METHOD FB_init : BOOL
VAR_INPUT
	bInitRetains : BOOL; // if TRUE, the retain variables are initialized (warm start / cold start)
	bInCopyCode : BOOL;  // if TRUE, the instance afterwards gets moved into the copy code (online change)
	stPTOStepperRef : POINTER TO ST_PTOStepperRef;
END_VAR
THIS^.pPTOStepperRef := stPTOStepperRef;
END_METHOD

PROPERTY P_bError : BOOL
GET
END_GET
END_PROPERTY

PROPERTY P_bIsActive : BOOL
GET
END_GET
END_PROPERTY

PROPERTY P_bIsLocked : BOOL
GET
P_bIsLocked := TRUE;
END_GET
END_PROPERTY

PROPERTY P_pPTOStepperRef : POINTER TO ST_PTOStepperRef
GET
P_pPTOStepperRef := pPTOStepperRef;
END_GET
END_PROPERTY

END_FUNCTION_BLOCK

// ---- Hardware/PTOStepper/FB_PTOStepperRotate.TcPOU
FUNCTION_BLOCK FB_PTOStepperRotate
VAR_INPUT
	bExecute	: BOOL;
	bStop		: BOOL;
	bCCW		: BOOL;	//Gegen Uhrzeiger
	nSpeed		: UINT;	//Steps/sec
END_VAR
VAR_OUTPUT
	bBusy		: BOOL;
END_VAR
VAR_IN_OUT
	pPTOStepperRef : POINTER TO ST_PTOStepperRef;
END_VAR
VAR
	nSpeedIntern : INT;
	nState : USINT;
END_VAR

IF bExecute THEN
	CASE nState OF
		0:	//Prepare
			IF bStop THEN
				RETURN;
			END_IF
			bBusy := TRUE;
			IF bCCW THEN
				nSpeedIntern := UINT_TO_INT(nSpeed);
			ELSE
				nSpeedIntern := -UINT_TO_INT(nSpeed);
			END_IF
			MEMCPY(ADR(pPTOStepperRef^.nFrequencyValue),ADR(nSpeedIntern),2);
			nState := 1;
			
		1:	//Waiting for stop
			IF bStop THEN
				pPTOStepperRef^.nFrequencyValue := 0;
				nState := 80;
				bBusy := FALSE;
			END_IF
	END_CASE
ELSE
	nState := 0;
	bBusy := FALSE;	
END_IF

END_FUNCTION_BLOCK

// ---- Hardware/PTOStepper/FB_PTOStepperMoveRel.TcPOU
FUNCTION_BLOCK FB_PTOStepperMoveRel
VAR_INPUT
	bExecute	: BOOL;
	bStop		: BOOL;
	nSteps		: INT;
	nSpeed		: UINT;	//Steps/sec	
END_VAR
VAR_OUTPUT
	bBusy		: BOOL;
END_VAR
VAR_IN_OUT
	pPTOStepperRef : POINTER TO ST_PTOStepperRef;	
END_VAR
VAR
	nState : USINT;
	nSpeedIntern: INT;
END_VAR

IF bExecute THEN
	CASE nState OF
		0:	//Prepare
			IF bStop THEN
				RETURN;
			END_IF
			
			bBusy := TRUE;
			IF nSteps < 0 THEN
				//CCW Drehung -> muss Richtung "0" drehen -> auf Counter "0" oder Counter underflow abfragen
				pPTOStepperRef^.nSetCounterValue := INT_TO_UINT(ABS(nSteps));
				nSpeedIntern := -UINT_TO_INT(nSpeed);
			ELSIF nSteps > 0 THEN
				//CW Drehung -> muss Richtung "0" drehen -> auf Counter >= SetCounter oder Counter overflow abfragen
				pPTOStepperRef^.nSetCounterValue := 0;
				nSpeedIntern := UINT_TO_INT(nSpeed);
			ELSE
				bBusy := FALSE;
				nState := 80;
				RETURN;
			END_IF
			pPTOStepperRef^.bSetCounter := TRUE;
			nState := 1;
			
		1:	//Start
			IF bStop THEN
				bBusy := FALSE;
				nState := 80;
				RETURN;
			END_IF
			IF pPTOStepperRef^.nSetCounterValue = pPTOStepperRef^.nCountervalue THEN
				pPTOStepperRef^.bSetCounter := FALSE;
				MEMCPY(ADR(pPTOStepperRef^.nFrequencyValue),ADR(nSpeedIntern),2);
				nState := 2;
			END_IF
			
		2:	//Waiting for target reached
			IF bStop OR
					 	//CCW Drehung -> abwärts zählen -> auf Counter "0" oder Counter underflow abfragen
						((nSteps < 0) AND ((pPTOStepperRef^.nCountervalue = 0) OR pPTOStepperRef^.bCounterUnderflow))
					 OR
					 	//CW Drehung -> aufwärts zählen -> auf Counter >= SetCounter oder Counter overflow abfragen
						((nSteps > 0) AND ((pPTOStepperRef^.nCountervalue >= INT_TO_UINT(ABS(nSteps))) OR pPTOStepperRef^.bCounterUnderflow))THEN
						
				pPTOStepperRef^.nFrequencyValue := 0;
				nState := 3;
			END_IF
			
		3:	//Wartezyklus
			bBusy := FALSE;
	END_CASE
ELSE
	nState := 0;
	bBusy := FALSE;
END_IF

END_FUNCTION_BLOCK

// ---- Hardware/MultiZ/Heater/FB_MzHeaterControl.TcPOU
FUNCTION_BLOCK FB_MzHeaterControl
VAR_INPUT
	bExecute 		: BOOL;
	nTempZone1		: UINT;		//Solltemperatur Heizzone 1
	nTempZone2		: UINT;		//Solltemperatur Heizzone 2
	nTempZone3		: UINT;		//Solltemperatur Heizzone 3
	bHeatingOn		: BOOL;		//Ein/Aus
END_VAR
VAR_OUTPUT
	bBusy : BOOL;
	bError : BOOL;
	nErrorId : ERRORID;	
END_VAR
VAR_IN_OUT
	pFbHeaterRef : POINTER TO FB_MZHeaterRef;
END_VAR
VAR
	fbSdoWrite		: FB_SDO_WRITE;
	fbSdoRead		: FB_SDO_Read;
	nState 			: USINT;
	nStateNext		: USINT;
END_VAR

IF pFbHeaterRef = 0 THEN
	RETURN;
END_IF

IF bExecute THEN
	IF nState = 0 THEN //Solltemperatur Zone 1 senden
		bBusy := TRUE;
		IF NOT bHeatingOn THEN	//keine Temperaturen senden
			nState := 3;
		ELSE
			pFbHeaterRef^.P_nTemp1Setpoint := nTempZone1;
			fbSdoWrite.nIndex := cTempSetPoint.nIndex;
			fbSdoWrite.nSubIndex := pFbHeaterRef^.nChannel;
			fbSdoWrite.nDataLength := cTempSetPoint.nLength;
			fbSdoWrite.nData := UINT_TO_DINT(nTempZone1);
			nState := 10;
			IF pFbHeaterRef^.pMultiZRef^.P_bLegacy THEN	//Heizzone2 und 3 nur bei Firmware ab V1.10.xx
				nStateNext := 3;
			ELSE
				nStateNext := 1;
			END_IF
		END_IF
	END_IF
	
	IF nState = 1 THEN //Solltemperatur Zone 2 senden
		fbSdoWrite.nIndex := cTempSetPoint2.nIndex;
		fbSdoWrite.nSubIndex := pFbHeaterRef^.nChannel;
		fbSdoWrite.nDataLength := cTempSetPoint2.nLength;
		fbSdoWrite.nData := UINT_TO_DINT(nTempZone2);
		nState := 10;
		nStateNext := 2;
	END_IF

	IF nState = 2 THEN //Solltemperatur Zone 3 senden
		fbSdoWrite.nIndex := cTempSetPoint3.nIndex;
		fbSdoWrite.nSubIndex := pFbHeaterRef^.nChannel;
		fbSdoWrite.nDataLength := cTempSetPoint3.nLength;
		fbSdoWrite.nData := UINT_TO_DINT(nTempZone3);
		nState := 10;
		nStateNext := 3;
	END_IF
	
	IF nState = 3 THEN //On/Off senden
		fbSdoWrite.nIndex := cHeatingOn.nIndex;
		fbSdoWrite.nSubIndex := pFbHeaterRef^.nChannel;
		fbSdoWrite.nDataLength := cHeatingOn.nLength;
		fbSdoWrite.nData := BOOL_TO_DINT(bHeatingOn);
		nState := 10;
		IF pFbHeaterRef^.P_bHeaterDetected THEN
			nStateNext := 80;
		ELSE
			nStateNext := 20;
		END_IF
		
	END_IF
	
	IF nState = 10 THEN
		fbSdoWrite(sADSNetID:= pFbHeaterRef^.pMultiZRef^.P_sAdsNetId, nPortNr:= pFbHeaterRef^.pMultiZRef^.P_nAdsPort, bExecute:= TRUE);		
		IF NOT fbSdoWrite.bBusy THEN
			IF fbSdoWrite.bError THEN
				bError := TRUE;
				bBusy := FALSE;
				nErrorId := fbSdoWrite.nAdsErrorId;
				nState := 99;
			ELSE
				nState := nStateNext;
				IF nState = 80 THEN
					bBusy := FALSE;
				END_IF
			END_IF
			fbSdoWrite(bExecute:= FALSE);
		END_IF
	ELSIF nState = 20 THEN //Das HeaterExist wird nur ausgelesen, wenn es nicht vorher schon in A_PrepareAxis im FB_MultiZRef erfolgt ist.
		//Dieser Fall tritt ein, wenn der Heizer später erst angesteckt wurde (Kartuschen-Halter und Piezo-Pipetten)
		fbSdoRead(sADSNetID:= pFbHeaterRef^.pMultiZRef^.P_sAdsNetId, nPortNr:= pFbHeaterRef^.pMultiZRef^.P_nAdsPort, nIndex:= cHeaterExist.nIndex, 
					nSubIndex:= pFbHeaterRef^.nChannel,	nDataLength:= cHeaterExist.nLength, bExecute:= TRUE);
		IF NOT fbSdoRead.bBusy THEN
			IF fbSdoRead.bError THEN
				bError := TRUE;
				bBusy := FALSE;
				nErrorId := fbSdoRead.nAdsErrorId;
				nState := 99;
			ELSE
				pFbHeaterRef^.P_bHeaterDetected := DINT_TO_BOOL(fbSdoRead.nData);
				nState := 80;
				bBusy := FALSE;
			END_IF
			fbSdoRead(bExecute:= FALSE);
		END_IF
	END_IF
ELSE
	nState := 0;
	bError := FALSE;
	nErrorId := 0;
END_IF

END_FUNCTION_BLOCK

// ---- Objects/Tools/FB_PassivPip.TcPOU
FUNCTION_BLOCK FB_PassivPip EXTENDS FB_GCodeTool IMPLEMENTS I_UsingDryPad, I_Dispenser
VAR_INPUT
END_VAR
VAR_OUTPUT
END_VAR
VAR
	//SpecProperties
	nDiluterObjId		: UINT;
	pDiluter			: POINTER TO FB_Diluter;
	pDiluter3Inputs		: POINTER TO FB_Diluter3Inputs;
	nDrypadArea			: USINT;
	tDryTime			: TIME;
	nDispFlowFix		: DINT;	//wird für das Dispensen benutzt, wenn Tool am HybridDispenser oder M127 (UniDispense)

	//****************************************Aktionvariablen****************************************************
	stActionDataSpec	: ST_ActionData;
	
	//Action: "Aspirate"
	bAspirate			: BOOL;
	nStateA_Aspirate	: USINT;
	nQuantity			: DINT;
	nFlow				: DINT;
	
	//Action: "Dispense"
	bDispense			: BOOL;
	nStateA_Dispense	: USINT;
	nDilInput			: USINT;
	bEndless			: BOOL;
	
	//Action: "DilMovePlunger"
	bDilMovePlunger		: BOOL;
	nStateA_DilMovePlunger	: USINT;
	nDilMovePlungerPos	: DINT;
	nDilMovePlungerSpeed: DINT;
	nDilMovePlungerValve: DINT;
	
	
	//Action: "Mix"
	bMix				: BOOL;
	nStateA_Mix			: USINT;
	nFlowAsp			: DINT;
	nFlowDisp			: DINT;
	nMixRepeats			: UINT;
	nCurrMixRepeats		: UINT;
	tMixDelay1			: TIME; //Delay zwischen Asp und Disp
	tMixDelay2			: TIME; //Delay nach jedem Zyklus
	timerMix			: TON;
	
	//Action: "Eject"
	bEject				: BOOL;
	nStateA_Eject		: USINT;
	fbMultiZTipEjector	: FB_MultiZTipEjector;
	
END_VAR

IF eCurrentState = E_MachineState.MACHINESTATE_Active THEN
	
	IF bAspirate THEN
		A_Aspirate();
		IF nStateA_Aspirate >= 80 THEN
			IF nStateA_Aspirate >= 99 THEN
				fbErrorList.M_Add(stError);
				bError := TRUE;	
			END_IF
			bAspirate := FALSE;
			nStateA_Aspirate := 0;
			M_RemoveListEntry(nSearchValue:= E_Action.ACTION_Aspirate);
		END_IF
	END_IF

	IF bDispense THEN
		A_Dispense();
		IF nStateA_Dispense >= 80 THEN
			IF nStateA_Dispense >= 99 THEN
				stError.Cmd := E_Action.ACTION_Dispense;
				fbErrorList.M_Add(stError);
				bError := TRUE;	
			END_IF
			bDispense := FALSE;
			nStateA_Dispense := 0;
			M_RemoveListEntry(nSearchValue:= E_Action.ACTION_Dispense);
		END_IF
	END_IF
	
	IF bMix THEN
		A_Mix();
		IF nStateA_Mix >= 80 THEN
			IF nStateA_Mix >= 99 THEN
				stError.Cmd := E_Action.ACTION_Mix;
				fbErrorList.M_Add(stError);
				bError := TRUE;	
			END_IF
			bMix := FALSE;
			nStateA_Mix := 0;
			M_RemoveListEntry(nSearchValue:= E_Action.ACTION_Mix);
		END_IF
	END_IF
	
	IF bEject THEN
		A_Eject();
		IF nStateA_Eject >= 80 THEN
			IF nStateA_Eject >= 99 THEN
				stError.Cmd := E_Action.ACTION_Eject;
				fbErrorList.M_Add(stError);
				bError := TRUE;	
			END_IF
			bEject := FALSE;
			nStateA_Eject := 0;
			M_RemoveListEntry(nSearchValue:= E_Action.ACTION_Eject);
		END_IF
	END_IF
	
	IF bDilMovePlunger THEN
		A_DilMovePlunger();
		IF nStateA_DilMovePlunger >= 80 THEN
			IF nStateA_DilMovePlunger >= 99 THEN
				stError.Cmd := E_Action.ACTION_DilMovePlunger;
				fbErrorList.M_Add(stError);
				bError := TRUE;	
			END_IF
			bDilMovePlunger := FALSE;
			nStateA_DilMovePlunger := 0;
			M_RemoveListEntry(nSearchValue:= E_Action.ACTION_DilMovePlunger);
		END_IF
	END_IF

END_IF

SUPER^();	//FB_MzTool aufrufen

aObjProcData[nNotifyId] := stProcessData;
stProcessData.n32Data[7] := BOOL_TO_DINT(bAspirate OR bDispense);

ACTION A_Aspirate:
IF pDiluter^.P_bError THEN
	stError.ErrorId := pDiluter^.P_nErrorId;
	stError.POUState := nStateA_Aspirate;
	nStateA_Aspirate := 99;
END_IF

CASE nStateA_Aspirate OF
	0:	MEMSET(ADR(stActionDataSpec),0,SIZEOF(stActionDataSpec));
		stActionDataSpec.eAction := E_Action.ACTION_DilPump;
		stActionDataSpec.aParams[1] := E_DilPumpMode.MODE_Suck;
		stActionDataSpec.aParams[2] := nQuantity; 
		stActionDataSpec.aParams[3] := nFlow;
		//stActionDataSpec.aParams[4]  //ReloadSpeed wird von DilConfig übernommen
		(*Beim normalen Diluter wird ValvePosReload aus der DilConfig übernommen, beim Diluter3Inputs wird
		die ValvePos über die InputNr ermittelt.*)
		IF pDiluter3Inputs > 0 THEN
			stActionDataSpec.aParams[6] := pDiluter3Inputs^.M_GetValvePosInput(nDilInput);
		END_IF
		
		stError.ErrorId := pDiluter^.M_ExeAction(stActionDataSpec);
		IF stError.ErrorId > 0 THEN
			stError.POUState := nStateA_Aspirate;
			nStateA_Aspirate := 99;
		ELSE
			nStateA_Aspirate := 1;	
		END_IF
		
	1:	//Warten bis Aspiration fertig
		IF NOT pDiluter^.M_GetActionBusy(E_Action.ACTION_DilPump) THEN
			nStateA_Aspirate := 80;
		END_IF
		
	70:	//Abbrechen
		MEMSET(ADR(stActionDataSpec),0,SIZEOF(stActionDataSpec));
		stActionDataSpec.eAction := E_Action.ACTION_Stop;
		
		pDiluter^.M_ExeAction(stActionDataSpec);
		nStateA_Aspirate := 71;
		
	71:	
		IF NOT pDiluter^.P_bBusy THEN
			nStateA_Aspirate := 80;
		END_IF
END_CASE

//Errorhandling
IF nStateA_Aspirate = 99 THEN
	stError.Cmd := E_Action.ACTION_Aspirate;
	stError.POU := E_POU.POU_FB_PassivPip;
	stError.POUAction := E_POUACT.POUACT_A_Aspirate;
	fbErrorList.M_Add(stError);
END_IF
END_ACTION

ACTION A_DilMovePlunger:
IF pDiluter^.P_bError THEN
	stError.ErrorId := pDiluter^.P_nErrorId;
	stError.POUState := nStateA_DilMovePlunger;
	nStateA_DilMovePlunger := 99;
END_IF

CASE nStateA_DilMovePlunger OF
	0:	MEMSET(ADR(stActionDataSpec),0,SIZEOF(stActionDataSpec));
		stActionDataSpec.eAction := E_Action.ACTION_DilMovePlunger;
		stActionDataSpec.aParams[1] := nDilMovePlungerPos;
		stActionDataSpec.aParams[2] := nDilMovePlungerSpeed;
		stActionDataSpec.aParams[3] := nDilMovePlungerValve;
		stError.ErrorId := pDiluter^.M_ExeAction(stActionDataSpec);
		IF stError.ErrorId > 0 THEN
			nStateA_DilMovePlunger := 99;
		ELSE
			nStateA_DilMovePlunger := 1;	
		END_IF
	
	1:	IF NOT pDiluter^.M_GetActionBusy(E_Action.ACTION_DilMovePlunger) THEN
			nStateA_DilMovePlunger := 80;
		END_IF
 		
	70: //Abrechen
		MEMSET(ADR(stActionDataSpec),0,SIZEOF(stActionDataSpec));
		stActionDataSpec.eAction := E_Action.ACTION_Stop;
		
		pDiluter^.M_ExeAction(stActionDataSpec);
		nStateA_DilMovePlunger := 71;
		
	71:	IF NOT pDiluter^.P_bBusy THEN
			nStateA_DilMovePlunger := 80;
		END_IF	
END_CASE

//Errorhandling
IF nStateA_DilMovePlunger = 99 THEN
	stError.Cmd := E_Action.ACTION_DilMovePlunger;
	stError.POU := E_POU.POU_FB_PassivPip;
	stError.POUAction := E_POUACT.POUACT_A_MovePlunger;
	fbErrorList.M_Add(stError);
END_IF
END_ACTION

ACTION A_Dispense:
IF pDiluter^.P_bError THEN
	stError.ErrorId := pDiluter^.P_nErrorId;
	stError.POUState := nStateA_Dispense;
	nStateA_Dispense := 99;
END_IF

CASE nStateA_Dispense OF
	0:	MEMSET(ADR(stActionDataSpec),0,SIZEOF(stActionDataSpec));
		stActionDataSpec.eAction := E_Action.ACTION_DilPump;
		stActionDataSpec.aParams[1] := E_DilPumpMode.MODE_Press;
		stActionDataSpec.aParams[2] := nQuantity; 
		stActionDataSpec.aParams[3] := nFlow;
		//stActionDataSpec.aParams[4]  //ReloadSpeed wird von DilConfig übernommen
		(*Beim normalen Diluter wird ValvePosReload aus der DilConfig übernommen, beim Diluter3Inputs wird
		die ValvePos über die InputNr ermittelt.*)
		IF pDiluter3Inputs > 0 THEN
			stActionDataSpec.aParams[6] := pDiluter3Inputs^.M_GetValvePosInput(nDilInput);
		END_IF
		stActionDataSpec.aParams[7] := BOOL_TO_DINT(bEndless);
		bEndless := FALSE;
		
		stError.ErrorId := pDiluter^.M_ExeAction(stActionDataSpec);
		IF stError.ErrorId > 0 THEN
			stError.POUState := nStateA_Dispense;
			nStateA_Dispense := 99;
		ELSE
			nStateA_Dispense := 1;	
		END_IF
		
	1:	//Warten bis Dispensen fertig
		IF NOT pDiluter^.M_GetActionBusy(E_Action.ACTION_DilPump) THEN
			nStateA_Dispense := 80;
		END_IF
		
	70:	//Abbrechen
		MEMSET(ADR(stActionDataSpec),0,SIZEOF(stActionDataSpec));
		stActionDataSpec.eAction := E_Action.ACTION_Stop;
		
		pDiluter^.M_ExeAction(stActionDataSpec);
		nStateA_Dispense := 71;
		
	71:	
		IF NOT pDiluter^.P_bBusy THEN
			nStateA_Dispense := 80;
		END_IF
END_CASE

//Errorhandling
IF nStateA_Dispense = 99 THEN
	stError.Cmd := E_Action.ACTION_Dispense;
	stError.POU := E_POU.POU_FB_PassivPip;
	stError.POUAction := E_POUACT.POUACT_A_Dispense;
	fbErrorList.M_Add(stError);
END_IF
END_ACTION

ACTION A_Eject:
fbMultiZTipEjector(pfbZAxisRef:= pZAxisRef, bExecute:= TRUE);

IF NOT fbMultiZTipEjector.bBusy THEN
	IF fbMultiZTipEjector.bError THEN
		stError.Cmd := E_Action.ACTION_Eject;
		stError.ErrorId := fbMultiZTipEjector.nErrorId;
		stError.POUState := nStateA_Eject;
		stError.POU := E_POU.POU_FB_PassivPip;
		stError.POUAction := E_POUACT.POUACT_A_Eject;
		fbErrorList.M_Add(stError);
		nStateA_Eject := 99;
	ELSE
		nStateA_Eject := 80;
	END_IF
	fbMultiZTipEjector(bExecute:= FALSE);
END_IF
END_ACTION

ACTION A_Mix:
IF pDiluter^.P_bError THEN
	stError.ErrorId := pDiluter^.P_nErrorId;
	stError.POUState := nStateA_Mix;
	nStateA_Mix := 99;
END_IF

CASE nStateA_Mix OF
	0:	//Aspirieren
		MEMSET(ADR(stActionDataSpec),0,SIZEOF(stActionDataSpec));
		stActionDataSpec.eAction := E_Action.ACTION_DilPump;
		stActionDataSpec.aParams[1] := E_DilPumpMode.MODE_Suck;
		stActionDataSpec.aParams[2] := nQuantity; 
		stActionDataSpec.aParams[3] := nFlowAsp;
		//stActionDataSpec.aParams[4]  //ReloadSpeed wird von DilConfig übernommen
		(*Beim normalen Diluter wird ValvePosReload aus der DilConfig übernommen, beim Diluter3Inputs wird
		die ValvePos über die InputNr ermittelt.*)
		IF pDiluter3Inputs > 0 THEN
			stActionDataSpec.aParams[6] := pDiluter3Inputs^.M_GetValvePosInput(nDilInput);
		END_IF
		
		stError.ErrorId := pDiluter^.M_ExeAction(stActionDataSpec);
		IF stError.ErrorId > 0 THEN
			stError.POUState := nStateA_Mix;
			nStateA_Mix := 99;
		ELSE
			nStateA_Mix := 1;	
		END_IF
		
	1:	//Aspirieren fertig?
		IF NOT pDiluter^.M_GetActionBusy(E_Action.ACTION_DilPump) THEN
			timerMix(IN:= TRUE, PT:= tMixDelay1);
			nStateA_Mix := 2;
		END_IF
		
	2:	//Timer?
		timerMix();
		IF timerMix.Q THEN
			timerMix(IN:= FALSE);
			nStateA_Mix := 3;
		END_IF
		
	3:	//Dispensen
		MEMSET(ADR(stActionDataSpec),0,SIZEOF(stActionDataSpec));
		stActionDataSpec.eAction := E_Action.ACTION_DilPump;
		stActionDataSpec.aParams[1] := E_DilPumpMode.MODE_Press;
		stActionDataSpec.aParams[2] := nQuantity; 
		stActionDataSpec.aParams[3] := nFlowDisp;
		//stActionDataSpec.aParams[4]  //ReloadSpeed wird von DilConfig übernommen
		(*Beim normalen Diluter wird ValvePosReload aus der DilConfig übernommen, beim Diluter3Inputs wird
		die ValvePos über die InputNr ermittelt.*)
		IF pDiluter3Inputs > 0 THEN
			stActionDataSpec.aParams[6] := pDiluter3Inputs^.M_GetValvePosInput(nDilInput);
		END_IF
		
		
		stError.ErrorId := pDiluter^.M_ExeAction(stActionDataSpec);
		IF stError.ErrorId > 0 THEN
			stError.POUState := nStateA_Mix;
			nStateA_Mix := 99;
		ELSE
			nStateA_Mix := 4;
		END_IF
		
	4:	//Dispensen fertig?
		IF NOT pDiluter^.M_GetActionBusy(E_Action.ACTION_DilPump) THEN
			nCurrMixRepeats := nCurrMixRepeats + 1;
			IF nCurrMixRepeats = nMixRepeats THEN
				nStateA_Mix := 80;
			ELSE
				timerMix(IN:= TRUE, PT:= tMixDelay2);
				nStateA_Mix := 5;
			END_IF
		END_IF
		
	5:	//Timer?
		timerMix();
		IF timerMix.Q THEN
			timerMix(IN:= FALSE);
			nStateA_Mix := 0;
		END_IF

	70:	//Abbrechen
		timerMix(IN:= FALSE);
		MEMSET(ADR(stActionDataSpec),0,SIZEOF(stActionDataSpec));
		stActionDataSpec.eAction := E_Action.ACTION_Stop;
		pDiluter^.M_ExeAction(stActionDataSpec);
		nStateA_Mix := 71;
		
	71:	IF NOT pDiluter^.P_bBusy THEN
			nStateA_Mix := 80;
		END_IF		
END_CASE

//Errorhandling
IF nStateA_Mix = 99 THEN
	stError.Cmd := E_Action.ACTION_Mix;
	stError.POU := E_POU.POU_FB_PassivPip;
	stError.POUAction := E_POUACT.POUACT_A_Mix;
	fbErrorList.M_Add(stError);
END_IF
END_ACTION

ACTION A_Reset:
//Ist noch eine Aktion aktiv?
IF nStateA_ResetSpec = 0 THEN 
	IF bAspirate THEN
		bAspirate := FALSE;
		nStateA_Aspirate := 0;
	END_IF

	IF bDispense THEN
		bDispense := FALSE;
		nStateA_Dispense := 0;
	END_IF
	
	IF bEject THEN
		bEject := FALSE;
		nStateA_Eject := 0;
	END_IF
	
	nStateA_ResetSpec := 80;
END_IF

SUPER^.A_Reset();
END_ACTION

ACTION A_Stop:
IF nStateA_Stop = 0 THEN
	
	IF bAspirate AND nStateA_Aspirate < 70 THEN
		nStateA_Aspirate := 70;
	END_IF
	
	IF bDispense AND nStateA_Dispense < 70 THEN
		nStateA_Dispense := 70;
	END_IF
	
	IF bMix AND nStateA_Mix < 70 THEN
		nStateA_Mix := 70;
	END_IF
	
	nStateA_Stop := 1;
END_IF

SUPER^.A_Stop();
END_ACTION

METHOD FB_init : BOOL
VAR_INPUT
	bInitRetains : BOOL; // if TRUE, the retain variables are initialized (warm start / cold start)
	bInCopyCode : BOOL;  // if TRUE, the instance afterwards gets moved into the copy code (online change)
END_VAR
eObjectType := E_ObjectType.OBJECTTYPE_PassivPip;
eObjectGroup := E_ObjectGroup.OBJECTGROUP_MzTool OR E_ObjectGroup.OBJECTGROUP_Device;
END_METHOD

METHOD M_AddChild : ERRORID
VAR_INPUT
	pObject : POINTER TO FB_Object;
	nSlotNr	: UINT;
	nIndex 	: INT;
END_VAR
//PassivePip kann folgende Objekt-Typen aufnehmen
//Needle, Tip, Nozzle
IF pObject > 0 THEN
	IF pObject^.P_eObjectType = E_ObjectType.OBJECTTYPE_Needle OR
		pObject^.P_eObjectType = E_ObjectType.OBJECTTYPE_Nozzle OR
		pObject^.P_eObjectType = E_ObjectType.OBJECTTYPE_Tip THEN
		M_AddChild := SUPER^.M_AddChild(pObject,nSlotNr,nIndex);
	ELSE
		M_AddChild := E_ErrorIdObjMgmt.ERRORID_InvalidParentObject;
	END_IF
ELSE
	M_AddChild := E_ErrorIdObjMgmt.ERRORID_InvalidParentObject;
END_IF
END_METHOD

METHOD M_CancelAction
VAR_INPUT
	eAction : E_Action;
END_VAR
CASE eAction OF
	E_Action.ACTION_Aspirate:
		IF bAspirate AND nStateA_Aspirate < 70 THEN
			nStateA_Aspirate := 70;
		END_IF
	E_Action.ACTION_Dispense:
		IF bDispense AND nStateA_Dispense < 70 THEN
			nStateA_Dispense := 70;
		END_IF
	E_Action.ACTION_Mix:
		IF bMix AND nStateA_Mix < 70 THEN
			nStateA_Mix := 70;
		END_IF	
ELSE
	SUPER^.M_CancelAction(eAction);
END_CASE
END_METHOD

METHOD M_CheckAction : ERRORID
VAR_INPUT
	refActionData 	: REFERENCE TO ST_ActionData;
	pCorrelObject	: POINTER TO FB_Object;
END_VAR

VAR
	pTarget : POINTER TO FB_TargetBase;
	pRack	: POINTER TO FB_Rack;
	pSlot	: POINTER TO FB_PieceSlot;	
END_VAR
CASE refActionData.eAction OF
	E_Action.ACTION_GetPipSample,
	E_Action.ACTION_MeasureTool,
	E_Action.ACTION_Dispense, //BasicAction für ActionOnArray
	E_Action.ACTION_Aspirate, //BasicAction für ActionOnArray
	E_Action.ACTION_Mix, //BasicAction für ActionOnArray
	E_Action.ACTION_TeachTarget:
		RETURN;
	E_Action.ACTION_WashTool:
		//Washmode checken
		IF refActionData.aParams[2] = E_WashMode.MODE_WashInside THEN
			M_CheckAction := M_CheckBottles();
		ELSIF refActionData.aParams[2] = E_WashMode.MODE_WashOutside THEN
			;
		ELSIF refActionData.aParams[2] = E_WashMode.MODE_WashInOutside THEN
			M_CheckAction := M_CheckBottles();
		ELSIF refActionData.aParams[2] = E_WashMode.MODE_DryOutside THEN
			;
		ELSE
			M_CheckAction := E_ErrorIdCmd.ERRORID_InvalidWashMode;	
		END_IF
	E_Action.ACTION_InsertTool:
		//PassivPip darf nur in offene Vials eintauchen
		//-> Target muss also ein VialRack sein (Reaktor nicht möglich, da Pip nicht von der Tiefe hinein passt)
		pTarget := pCorrelObject;
		IF pTarget > 0 THEN
			IF (pTarget^.P_eObjectGroup AND E_ObjectGroup.OBJECTGROUP_Rack) = E_ObjectGroup.OBJECTGROUP_Rack THEN
				pRack := pTarget;
				pSlot := pRack^.M_GetSlot(DINT_TO_UINT(refActionData.aParams[2]));
				IF pSlot > 0 THEN
					IF pSlot^.P_pPiece = 0 THEN
						M_CheckAction := E_ErrorIdCmd.ERRORID_NoPieceInSlot;
						RETURN;
					ELSIF NOT (pSlot^.P_pPiece^.P_eObjectType = E_ObjectType.OBJECTTYPE_Vial OR pSlot^.P_pPiece^.P_eObjectType = E_ObjectType.OBJECTTYPE_FlipTube) THEN
						M_CheckAction := E_ErrorIdCmd.ERRORID_InvalidPieceType;
					END_IF
				ELSE
					M_CheckAction := E_ErrorIdCmd.ERRORID_InvalidTargetSlot;
					RETURN;
				END_IF	
			ELSE
				M_CheckAction := E_ErrorIdCmd.ERRORID_UnsuitableTarget;	
			END_IF
		ELSE
			M_CheckAction := E_ErrorIdCmd.ERRORID_UnsuitableTarget;	
		END_IF	
ELSE
	M_CheckAction := SUPER^.M_CheckAction(refActionData, pCorrelObject);
END_CASE
END_METHOD

METHOD M_CheckBottles : ERRORID
VAR_INPUT
END_VAR
IF pDiluter > 0 THEN
	M_CheckBottles := pDiluter^.M_CheckBottles(0);
END_IF
END_METHOD

METHOD M_CheckGCodeStart : ERRORID
VAR_INPUT
END_VAR
IF NOT (P_bIsInit AND pDiluter^.P_bIsInit) THEN
	M_CheckGCodeStart := E_ErrorIdCmd.ERRORID_DeviceNotInitialized;
END_IF
END_METHOD

METHOD M_CheckProps : ERRORID
VAR_INPUT
END_VAR
M_CheckProps := SUPER^.M_CheckProps();
IF M_CheckProps > 0 THEN
	RETURN;
END_IF
//Konfigurierte Properties checken
//zugeordneter Diluter
IF pDiluter = 0 THEN
	M_CheckProps := E_ErrorIdObjMgmt.ERRORID_InvalidDiluterObjId; //Error
	RETURN;
END_IF

IF nNumberOfSlots > 0 AND_THEN pPiece = 0 THEN
	M_CheckProps := E_ErrorIdObjMgmt.ERRORID_NoNozzleOnTool;
END_IF
END_METHOD

METHOD M_DispenserPrepare : ERRORID
VAR_INPUT
END_VAR
IF NOT (eCurrentState = E_MachineState.MACHINESTATE_Idle OR
	eCurrentState = E_MachineState.MACHINESTATE_Active OR
	eCurrentState = E_MachineState.MACHINESTATE_Ready) THEN
	M_DispenserPrepare := E_ErrorIdCmd.ERRORID_InvalidState;
	RETURN;
END_IF

IF bAspirate OR bDispense OR bMix OR bDilMovePlunger THEN
	M_DispenserPrepare := E_ErrorIdCmd.ERRORID_BasicActionActive;
ELSE
	//Welche Bottle muss den hier überprüft werden?
	M_DispenserPrepare := pDiluter^.M_CheckBottles(0);
	IF M_DispenserPrepare > 0 THEN
		RETURN;
	END_IF
	//Diluter auf Ausgangsposition (unten) fahren
	nDilMovePlungerPos := 24000;
	nDilMovePlungerSpeed := pDiluter^.P_nConfigReloadSpeed;
	nDilMovePlungerValve := pDiluter^.P_nValvePosInput;
	fbList.A_AddHeadValue(hList := hList, putValue := E_Action.ACTION_DilMovePlunger);
	bDilMovePlunger := TRUE;
	bBusy := TRUE;
	eCurrentState := E_MachineState.MACHINESTATE_Active;
END_IF
END_METHOD

METHOD M_DispenserStart : ERRORID
VAR_INPUT
END_VAR
IF NOT (eCurrentState = E_MachineState.MACHINESTATE_Idle OR
	eCurrentState = E_MachineState.MACHINESTATE_Active OR
	eCurrentState = E_MachineState.MACHINESTATE_Ready) THEN
	M_DispenserStart := E_ErrorIdCmd.ERRORID_InvalidState;
	RETURN;
END_IF

IF bAspirate OR bDispense OR bMix THEN
	M_DispenserStart := E_ErrorIdCmd.ERRORID_BasicActionActive;
ELSE //Ein
	nFlow := nDispFlowFix;
	nQuantity := 0;
	bEndless := TRUE;
	fbList.A_AddHeadValue(hList := hList, putValue := E_Action.ACTION_Dispense);
	bDispense := TRUE;
	bBusy := TRUE;
	eCurrentState := E_MachineState.MACHINESTATE_Active;		
END_IF
END_METHOD

METHOD M_DispenserStop : ERRORID
VAR_INPUT
END_VAR
//Achtung, hier kann es sein, dass noch im PrepareModus!
M_CancelAction(E_Action.ACTION_Dispense);
END_METHOD

METHOD M_ExeAction : ERRORID
VAR_INPUT
	refActionData : REFERENCE TO ST_ActionData;	
END_VAR
IF NOT (eCurrentState = E_MachineState.MACHINESTATE_Idle OR
	eCurrentState = E_MachineState.MACHINESTATE_Active OR
	eCurrentState = E_MachineState.MACHINESTATE_Ready) THEN
	M_ExeAction := E_ErrorIdCmd.ERRORID_InvalidState;
	RETURN;
END_IF

CASE refActionData.eAction OF
		
	E_Action.ACTION_Aspirate:
		IF NOT bAspirate THEN
			nQuantity := refActionData.aParams[1];
			nFlow := refActionData.aParams[2];
			IF pDiluter3Inputs > 0 THEN //Beim Diluter3Inputs wird die ValvePos für den entsprechnenden Input aus dem Diluter geholt.
				nDilInput := DINT_TO_USINT(refActionData.aParams[3]);
				IF nDilInput < 1 OR nDilInput > 3 THEN
					M_ExeAction := E_ErrorIdCmd.ERRORID_InvalidDiluterInput;
					RETURN;
				END_IF
			ELSE
				nDilInput := 0;
			END_IF
			M_ExeAction := pDiluter^.M_CheckBottles(nDilInput); //Checken, ob Bottles OK
			IF M_ExeAction > 0 THEN
				RETURN;
			END_IF			
			fbList.A_AddHeadValue( hList := hList, putValue := E_Action.ACTION_Aspirate);
			bAspirate := TRUE;
		END_IF
		
	E_Action.ACTION_Dispense:
		IF NOT bDispense THEN
			nQuantity := refActionData.aParams[1];
			nFlow := refActionData.aParams[2];
			IF pDiluter3Inputs > 0 THEN //Beim Diluter3Inputs wird die ValvePos für den entsprechnenden Input aus dem Diluter geholt.
				nDilInput := DINT_TO_USINT(refActionData.aParams[3]);
				IF nDilInput < 1 OR nDilInput > 3 THEN
					M_ExeAction := E_ErrorIdCmd.ERRORID_InvalidDiluterInput;
					RETURN;
				END_IF
			ELSE
				nDilInput := 0;
			END_IF
			M_ExeAction := pDiluter^.M_CheckBottles(nDilInput); //Checken, ob Bottles OK
			IF M_ExeAction > 0 THEN
				RETURN;
			END_IF			
			fbList.A_AddHeadValue(hList := hList, putValue := E_Action.ACTION_Dispense);
			bDispense := TRUE;
		END_IF
		
	E_Action.ACTION_Mix:
		IF NOT bMix THEN
			M_ExeAction := pDiluter^.M_CheckBottles(0); //Checken, ob Bottles OK
			IF M_ExeAction > 0 THEN
				RETURN;
			END_IF			
			nQuantity := refActionData.aParams[1];
			nFlowAsp := refActionData.aParams[2];
			nFlowDisp := refActionData.aParams[3];
			nMixRepeats := DINT_TO_UINT(refActionData.aParams[4]);
			nCurrMixRepeats := 0;
			tMixDelay1 := DINT_TO_TIME(refActionData.aParams[5]);
			tMixDelay2 := DINT_TO_TIME(refActionData.aParams[6]);
			nDilInput := DINT_TO_USINT(refActionData.aParams[7]);
			fbList.A_AddHeadValue(hList := hList, putValue := E_Action.ACTION_Mix);
			bMix := TRUE;
		END_IF
		
	E_Action.ACTION_Eject:
		//TipEjector vorhanden??
		IF pZAxisRef^.eFixedToolType <> E_MzToolType.TOOL_TYPE_TipEjector THEN
			M_ExeAction := E_ErrorIdCmd.ERRORID_ToolHasNoEjector;
			RETURN;	
		END_IF
		
		IF NOT bEject THEN
			fbList.A_AddHeadValue(hList := hList, putValue := E_Action.ACTION_Eject);
			bEject := TRUE;
		END_IF
			
	E_Action.ACTION_MoveX,E_Action.ACTION_MoveY,E_Action.ACTION_MoveXY:
		IF pZAxisRef^.stInput.nToolState.1 THEN
			M_ExeAction := ERRORID_PipMoveWithZSensor;  //Error
		ELSE
			M_ExeAction := SUPER^.M_ExeAction(refActionData);
			RETURN;	
		END_IF

	E_Action.ACTION_MoveZ:
		IF pZAxisRef^.stInput.nToolState.1 THEN
			eMoveModeZ := DINT_TO_USINT(refActionData.aParams[1]);
			IF NOT(eMoveModeZ = E_MoveMode.MODE_Free OR eMoveModeZ = E_MoveMode.MODE_Home) THEN
				M_ExeAction := ERRORID_PipMoveWithZSensor;  //Error
			END_IF
		ELSE
			M_ExeAction := SUPER^.M_ExeAction(refActionData);
			RETURN;	
		END_IF
		
	ELSE
		M_ExeAction := SUPER^.M_ExeAction(refActionData);
		RETURN;
END_CASE

bBusy := TRUE;
eCurrentState := E_MachineState.MACHINESTATE_Active;
END_METHOD

METHOD M_GetAllProps : ERRORID
VAR_INPUT
	refCmdData : REFERENCE TO  ST_CmdData;
END_VAR
//BaseProperties lesen
SUPER^.M_GetAllProps(refCmdData);

nCurrentPropIndex := nCurrentPropIndex + 1;
refCmdData.n32Data[nCurrentPropIndex] := nDiluterObjId;
nCurrentPropIndex := nCurrentPropIndex + 1;
refCmdData.n32Data[nCurrentPropIndex] := nDrypadArea;
nCurrentPropIndex := nCurrentPropIndex + 1;
refCmdData.n32Data[nCurrentPropIndex] := TIME_TO_DINT(tDryTime);
//TipEjector exist
nCurrentPropIndex := nCurrentPropIndex + 1;
IF pZAxisRef^.eFixedToolType = E_MzToolType.TOOL_TYPE_TipEjector THEN
	refCmdData.n32Data[nCurrentPropIndex] := 1;
ELSE
	refCmdData.n32Data[nCurrentPropIndex] := 0;
END_IF
nCurrentPropIndex := nCurrentPropIndex + 1;
refCmdData.n32Data[nCurrentPropIndex] := nDispFlowFix;
END_METHOD

METHOD M_SetAllProps : ERRORID
VAR_INPUT
	refCmdData : REFERENCE TO  ST_CmdData;
END_VAR

VAR
	pObject : POINTER TO FB_Object;
END_VAR
M_SetAllProps := SUPER^.M_SetAllProps(refCmdData);

IF M_SetAllProps > 0 THEN
	RETURN;
END_IF

pDiluter := 0;
pDiluter3Inputs := 0;
//Diluter
nCurrentPropIndex := nCurrentPropIndex + 1;
nSpecPropIndex := nCurrentPropIndex;
nDiluterObjId :=  DINT_TO_UINT(refCmdData.n32Data[nCurrentPropIndex]);
pObject := fbObjectDirectory.M_GetObjPointer(nDiluterObjId);
IF pObject > 0 THEN
	IF pObject^.P_eObjectType = E_ObjectType.OBJECTTYPE_Diluter THEN
		pDiluter := pObject;
	ELSIF pObject^.P_eObjectType = E_ObjectType.OBJECTTYPE_Diluter3Inputs THEN
		pDiluter := pObject;
		pDiluter3Inputs := pObject;
	ELSE
		M_SetAllProps := E_ErrorIdObjMgmt.ERRORID_InvalidDiluterObjId;
		RETURN;		
	END_IF
ELSE
	M_SetAllProps := E_ErrorIdObjMgmt.ERRORID_InvalidDiluterObjId;
	RETURN;	
END_IF

//DrypadArea
nCurrentPropIndex := nCurrentPropIndex + 1;
nDrypadArea := DINT_TO_USINT(refCmdData.n32Data[nCurrentPropIndex]);

//DryTime
nCurrentPropIndex := nCurrentPropIndex + 1;
tDryTime := DINT_TO_TIME(refCmdData.n32Data[nCurrentPropIndex]);

//TipEjector
nCurrentPropIndex := nCurrentPropIndex + 1;
IF refCmdData.n32Data[nCurrentPropIndex].0 THEN
	pZAxisRef^.eFixedToolType := E_MzToolType.TOOL_TYPE_TipEjector;
END_IF

//HybridDispFlow
nCurrentPropIndex := nCurrentPropIndex + 1;
nDispFlowFix := refCmdData.n32Data[nCurrentPropIndex];

nNoOfProps := nCurrentPropIndex + 1;
END_METHOD

METHOD M_SetPrintParams : ST_MethResult
VAR_INPUT
	eType 		: E_PrintParamType;
	nNumerator	: USINT;
	nValue		: DINT;
END_VAR
IF eType = E_PrintParamType.Flow THEN
	IF nNumerator <> 1 THEN
		M_SetPrintParams.bError := TRUE;
		M_SetPrintParams.nErrorId := E_ErrorIdCmd.ERRORID_InvalidPrintParamNumerator;
		RETURN;
	END_IF
	fbObjectDirectory.M_SetObjChange(nObjectID); //Info an GUI
	nDispFlowFix := nValue;
ELSE
	M_SetPrintParams.bError := TRUE;
	M_SetPrintParams.nErrorId := E_ErrorIdCmd.ERRORID_InvalidPrintParamType;
END_IF
END_METHOD

METHOD M_SetSingleProp : ERRORID
VAR_INPUT
	refCmdData : REFERENCE TO  ST_CmdData;
END_VAR
IF (nSpecPropIndex + 1) = refCmdData.aHeader[1] THEN	//DryPadArea
	nDrypadArea := DINT_TO_USINT(refCmdData.n32Data[0]);
ELSIF (nSpecPropIndex + 2) = refCmdData.aHeader[1] THEN //DryTime
	tDryTime := DINT_TO_TIME(refCmdData.n32Data[0]);
ELSIF (nSpecPropIndex + 4) = refCmdData.aHeader[1] THEN	//HybridDispFlow
	nDispFlowFix := refCmdData.n32Data[0];
ELSE
	M_SetSingleProp := SUPER^.M_SetSingleProp(refCmdData);
END_IF
END_METHOD

METHOD M_StartUniDispense : ERRORID
VAR_INPUT
	nParam1 : DINT; //Quantity
	nParam2 : DINT; //unused
END_VAR

VAR_OUTPUT
	bIsContinous : BOOL;
END_VAR

VAR
	stActionData : ST_ActionData;
END_VAR
IF nParam1 = 0 THEN
	bIsContinous := TRUE;
	bEndless := TRUE;
ELSE
	bEndless := FALSE;
END_IF

stActionData.aParams[1] := nParam1; //Quantitiy
stActionData.aParams[2] := nDispFlowFix;
stActionData.eAction := E_Action.ACTION_Dispense;
M_StartUniDispense := M_ExeAction(stActionData);
END_METHOD

METHOD M_StopUniDispense : ERRORID
VAR_INPUT
END_VAR
M_CancelAction(E_Action.ACTION_Dispense);
END_METHOD

PROPERTY P_bSensorMounted : BOOL
GET
P_bSensorMounted := pZAxisRef^.stInput.nToolState.1;
END_GET
END_PROPERTY

PROPERTY P_eDispenserState : E_DispenserState
GET
IF bDilMovePlunger THEN
	P_eDispenserState := E_DispenserState.Preparing;	
ELSIF bDispense THEN
	P_eDispenserState := E_DispenserState.Dispensing;
END_IF
END_GET
END_PROPERTY

PROPERTY P_nDrypadArea : USINT
GET
P_nDrypadArea := nDrypadArea;
END_GET
END_PROPERTY

PROPERTY P_pDiluter : POINTER TO FB_Diluter
GET
P_pDiluter := pDiluter;
END_GET
END_PROPERTY

PROPERTY P_rToolRadius : REAL
GET
VAR
	stDim : ST_3DDimension;
END_VAR
P_rToolRadius := 1500.0;
END_GET
END_PROPERTY

PROPERTY P_tDryTime : TIME
GET
P_tDryTime := tDryTime;
END_GET
END_PROPERTY

END_FUNCTION_BLOCK

// ---- Objects/Devices/FB_Diluter.TcPOU
FUNCTION_BLOCK FB_Diluter EXTENDS FB_Object IMPLEMENTS I_Device

VAR
	bInitFB				: BOOL := TRUE;			//zum erstmaligen Initialisieren des FB
	bError				: BOOL;
	stError				: ST_Error;
	bStopAllOnError		: BOOL;
	eCurrentState		: E_MachineState := E_MachineState.MACHINESTATE_Idle;
	nNotifyId			: UINT;
	nErrorId			: ERRORID;
	bCanceled			: BOOL;
	
	nParentSlotNr		: UINT;		//Diluter befindet sich zwar an keinem Slot, aber virtuell in der GUI (am Root)#
	
	//Specproperties
	nChannel			: USINT;	//Diluterkanal
	nSyringeSize		: DINT;		//Spritzengröße
	eReadedValveType	: E_DilValveType;
	
	nSysLiquidBottle 	: USINT;
	nWasteBottle 		: USINT;
	nConfigReloadSpeed	: DINT;
	eValveType			: E_DilValveType;
	nValvePosInput		: SINT;
	nValvePosOutput		: SINT;
	nValvePosWaste		: SINT;
	
	pDiluterRef1		: POINTER TO FB_HwRefDiluter;
	
	//Diluterbausteine
	fbGetPlungerPos		: FB_Dil_GetPlungerPos;
	fbGetValveConfig	: FB_Dil_GetValveConfig;
	fbSetValveConfig	: FB_Dil_SetValveConfig;
	fbGetValvePos		: FB_Dil_GetValvePos;
	fbInit				: FB_Dil_Init;
	fbTransfer 			: FB_Dil_Transfer;
	fbMoveValve			: FB_Dil_MoveValve;
	fbMoveToPos			: FB_Dil_MoveToPos;
	fbPump				: FB_Dil_Pump;
	fbStop				: FB_Dil_Stop;
	fbSendCmd			: FB_Dil_SendCmd(GVL_RS232.fbSerialPortDiluter);
	
	//****************************************Aktionvariablen****************************************************

	eCurrentAction		: E_Action;
	nStateAction		: USINT;
	//Action: "Init"
	bInit				: BOOL;
	bReInit				: BOOL;
	bFlagA_Init			: BOOL := TRUE;		//Hilfsflag A_Init()
	bIsInit				: BOOL;
	bValveConfigWritten : BOOL;

	//Action: "MovePlunger"
	bMovePlunger		: BOOL;
	
	//Action: "MoveValve"
	bMoveValve			: BOOL;
	
	//Action: "DilPump")
	bPump				: BOOL;
	bEndless			: BOOL;
	bFirstReload		: BOOL;
	
	//Action: "Transfer"
	bTransfer			: BOOL;
	nPreSteps			: INT;
	nPostSteps			: INT;
	pDilRefDest			: POINTER TO FB_Diluter;
	
	//Action: "Prepare"
	bPrepare			: BOOL;
	ePrepareMode		: E_DilPrepareMode;
	
	
	//Action: "DilStop"
	bStop				: BOOL;
	nStateA_Stop		: USINT;			//State von A_Stop()
	
	//gemeinsame Action-Parameter
	nStateNext			: USINT;
	ePumpMode			: E_DilPumpMode;
	nTotalSteps			: UDINT;	//Quantity in Microsteps
	nSpeedPump			: DINT;		//Geschwindigkeit Pumpen in Halbsteps/s
	nSpeedReload		: DINT;		//Geschwindigkeit Nachladen in Halbsteps/s
	nValvePosPump		: SINT;
	nValvePosReload		: SINT;
	nSetPosPlunger		: UINT;		//Kolbenposition aktuell

	nStateA_Reset		: USINT;	//State von A_Reset();
	stProcessData		: ST_ObjectProcData;
	
END_VAR

VAR_OUTPUT
	bBusy				: BOOL;
END_VAR

IF bInitFB THEN
	bInitFB := FALSE;
	//Fehlerstruktur vorausfüllen
	stError.HardwareGrp := E_HardwareGrp.Diluter;
	stError.POU := E_POU.POU_FB_Diluter;
END_IF

CASE eCurrentState OF
	E_MachineState.MACHINESTATE_Active:
		bBusy := TRUE;
		IF bInit THEN
			A_Init();
			IF nStateAction >= 80 THEN
				IF nStateAction >= 99 THEN
					bError := TRUE;	
				END_IF
				bInit := FALSE;
				nStateAction := 0;
			END_IF
		END_IF
		
		IF bMovePlunger THEN //Kolben bewegen
			A_MovePlunger();
			IF nStateAction >= 80 THEN
				IF nStateAction >= 99 THEN
					bError := TRUE;
				END_IF
				bMovePlunger := FALSE;
				nStateAction := 0;
			END_IF
		END_IF
		
		IF bMoveValve THEN	//Ventil stellen
			A_MoveValve();
			IF nStateAction >= 80 THEN
				IF nStateAction >= 99 THEN
					bError := TRUE;	
				END_IF
				bMoveValve := FALSE;
				nStateAction := 0;
			END_IF
		END_IF
		
		IF bPump THEN	//Pumpen
			A_Pump();
			IF nStateAction >= 80 THEN
				IF nStateAction >= 99 THEN
					bError := TRUE;	
				END_IF
				bPump := FALSE;
				nStateAction := 0;
			END_IF
		END_IF
		
		IF bTransfer THEN	//Transfer von Dil1 zu Dil2
			A_Transfer();
			IF nStateAction >= 80 THEN
				IF nStateAction >= 99 THEN
					bError := TRUE;	
				END_IF
				bTransfer := FALSE;
				nStateAction := 0;
			END_IF
		END_IF

		IF bPrepare THEN
			A_Prepare();
			IF nStateAction >= 80 THEN
				IF nStateAction >= 99 THEN
					bError := TRUE;	
				END_IF
				bPrepare := FALSE;
				nStateAction := 0;
			END_IF
		END_IF
 
 		IF bStop THEN
			A_Stop();
			IF nStateA_Stop >= 80 THEN
				IF nStateA_Stop >= 99 THEN
					bError := TRUE;	
				END_IF
				bStop := FALSE;
				nStateA_Stop := 0;
				nStateAction := 0;
			END_IF							
		END_IF
		
		IF NOT (bInit OR bMovePlunger OR bMoveValve OR bPump OR bTransfer OR bPrepare OR bStop) THEN
			eCurrentAction := E_Action.ACTION_Nothing;
			eCurrentState := E_MachineState.MACHINESTATE_Idle;
			bBusy := FALSE;
		END_IF

		IF bError THEN
			eCurrentAction := E_Action.ACTION_Nothing;
			eCurrentState := E_MachineState.MACHINESTATE_Error;
			bBusy := FALSE;
		END_IF

	E_MachineState.MACHINESTATE_Reset:
		A_Reset();
		IF nStateA_Reset = 80 THEN
			nStateAction := 0;
			nStateA_Stop := 0;
			nStateA_Reset := 0;
			bBusy := FALSE;
			bError := FALSE;
			bStopAllOnError := FALSE;
			stError.Cmd := 0;
			stError.ErrorId := 0;
			eCurrentState := E_MachineState.MACHINESTATE_Idle;
		ELSIF
			nStateA_Reset = 99 THEN
			fbErrorList.M_Add(stError);
			nStateA_Reset := 0;
			bBusy := FALSE;
			bError := TRUE;
			eCurrentState := E_MachineState.MACHINESTATE_Error;			
		END_IF
	
	E_MachineState.MACHINESTATE_Error:
		bBusy := FALSE;
END_CASE

IF pDiluterRef1 > 0 THEN
	bIsInit := pDiluterRef1^.bIsInit;
	stProcessData.n32Data[3] := pDiluterRef1^.nActValvePos;
	stProcessData.n32Data[4] := pDiluterRef1^.nActPlungerPos;
END_IF

//Prozessdaten aktualisieren
stProcessData.nObjId := nObjectID;
stProcessData.n32Data[0] := BOOL_TO_DINT(bIsInit);
stProcessData.n32Data[1] := eCurrentState;
stProcessData.n32Data[2] := stError.ErrorId;

aObjProcData[nNotifyId] := stProcessData;

ACTION A_Init:
stError.POUState := nStateAction;

IF nStateAction = 0 THEN
	IF pDiluterRef1 = 0 THEN
		nStateAction := 99;
	ELSE
		bValveConfigWritten := FALSE;		
		nStateAction := 1;
	END_IF
END_IF

CASE nStateAction OF
	1:	//ValveConfig lesen
		fbGetValveConfig(DilSendCmd:= fbSendCmd, pDilRef:= pDiluterRef1, bExecute := TRUE);
		IF NOT fbGetValveConfig.bBusy THEN
			IF fbGetValveConfig.bError THEN
				stError.ErrorId := fbGetValveConfig.nErrorId;
				nStateAction := 99;
			ELSE
				eReadedValveType := fbGetValveConfig.nValue;
				IF eReadedValveType <> eValveType THEN
					IF bValveConfigWritten THEN
						//Es wurde bereits versucht, die ValveConfig zu schreiben
						stError.ErrorId := E_ErrorIdDiluter.ERRORID_InvalidValveType;
						nStateAction := 99;
					ELSE
						//ValveConfig schreiben
						nStateAction := 2;
					END_IF
				ELSE
					IF bValveConfigWritten THEN
						nStateAction := 4; //In jedem Fall initialisieren
					ELSE
						nStateAction := 3;
					END_IF
				END_IF
			END_IF
			fbGetValveConfig(DilSendCmd:= fbSendCmd, pDilRef:= pDiluterRef1, bExecute := FALSE);
		END_IF
		
	2:	//ValveConfig schreiben
		fbSetValveConfig(DilSendCmd:= fbSendCmd, pDilRef:= pDiluterRef1, eValveType:= eValveType, bExecute := TRUE);
		IF NOT fbSetValveConfig.bBusy THEN
			IF fbSetValveConfig.bError THEN
				stError.ErrorId := fbGetValveConfig.nErrorId;
				nStateAction := 99;
			ELSE
				bValveConfigWritten := TRUE;
				nStateAction := 1; //nochmal auslesen
			END_IF
			fbSetValveConfig(DilSendCmd:= fbSendCmd, pDilRef:= pDiluterRef1, bExecute := FALSE);
		END_IF
		
	3:	//PlungerPos lesen, um festzustellen, ob Dil bereits initialisiert wurde
		fbGetPlungerPos(DilSendCmd:= fbSendCmd, pDilRef:= pDiluterRef1, bExecute := TRUE);
		IF NOT fbGetPlungerPos.bBusy THEN
			IF fbGetPlungerPos.bError THEN
				stError.ErrorId := fbGetPlungerPos.nErrorId;
				nStateAction := 99;
			ELSE
				IF pDiluterRef1^.nActPlungerPos = 0 OR bReInit THEN
					nStateAction := 4;
				ELSE
					nStateAction := 5;
				END_IF				
			END_IF
			fbGetPlungerPos(DilSendCmd:= fbSendCmd, pDilRef:= pDiluterRef1, bExecute := FALSE);
		END_IF

	4:	//Initialisieren
		fbInit(DilSendCmd:= fbSendCmd, pDilRef:= pDiluterRef1, bExecute := TRUE);
		IF NOT fbInit.bBusy THEN
			nStateAction := 5;
			IF fbInit.bError THEN
				stError.ErrorId := fbInit.nErrorId;
				nStateAction := 99;
			END_IF
			fbInit(DilSendCmd:= fbSendCmd, pDilRef:= pDiluterRef1, bExecute := FALSE);
		END_IF
		
	5:	//Plunger-Pos lesen (Ergebnis steht in pDilRef)
		fbGetPlungerPos(DilSendCmd:= fbSendCmd, pDilRef:= pDiluterRef1, bExecute := TRUE);
		IF NOT fbGetPlungerPos.bBusy THEN
			nStateAction := 6;
			IF fbGetPlungerPos.bError THEN
				stError.ErrorId := fbGetPlungerPos.nErrorId;
				nStateAction := 99;
			END_IF
			fbGetPlungerPos(DilSendCmd:= fbSendCmd, pDilRef:= pDiluterRef1, bExecute := FALSE);
		END_IF
		
	6:	//Valve-Pos lesen (Ergebnis steht in pDiluterRef1)
		fbGetValvePos(DilSendCmd:= fbSendCmd,pDilRef:= pDiluterRef1, bExecute := TRUE);
		IF NOT fbGetValvePos.bBusy THEN
			IF fbGetValvePos.bError THEN
				stError.ErrorId := fbGetValvePos.nErrorId;
				nStateAction := 99;
			ELSE
				pDiluterRef1^.bIsInit := TRUE;
				nStateAction := 80;	
			END_IF
			fbGetValvePos(DilSendCmd:= fbSendCmd, pDilRef:= pDiluterRef1, bExecute := FALSE);
		END_IF
END_CASE

//Errorhandling
IF nStateAction = 99 THEN
	stError.Cmd := E_Action.ACTION_Init;
	stError.POUAction := E_POUACT.POUACT_A_Init;
	fbErrorList.M_Add(stError);
END_IF
END_ACTION

ACTION A_MovePlunger:
stError.POUState := nStateAction;

CASE nStateAction OF
	0:	
		fbMoveToPos(nTopSpeed:= DINT_TO_UINT(nSpeedPump), nPosition:= nSetPosPlunger, 
					nValvePos:= nValvePosPump, bExecute:= TRUE, DilSendCmd:= fbSendCmd, pDilRef:= pDiluterRef1);

		IF NOT fbMoveToPos.bBusy THEN
			IF fbMoveToPos.bError THEN
				nStateAction := 99;
				stError.ErrorId := fbMoveToPos.nErrorId;
			ELSE
				
				nStateAction := 80;
			END_IF
			fbMoveToPos(bExecute:= FALSE, DilSendCmd:= fbSendCmd, pDilRef:= pDiluterRef1);			
		END_IF
		
	70:	//Abbrechen
		//Falls "fbMoveToPos" noch "Busy" dann "Abbrechen"
		IF fbMoveToPos.bBusy THEN
			fbMoveToPos(bExecute:= FALSE, DilSendCmd:= fbSendCmd, pDilRef:= pDiluterRef1);
		ELSE
			nStateAction := 71;	
		END_IF
		
	71:			
		fbStop(bExecute:= TRUE, DilSendCmd:= fbSendCmd);
		
		IF NOT fbStop.bBusy THEN
			IF fbStop.bError THEN
				nStateAction := 99;
				stError.ErrorId := fbStop.nErrorId;
			ELSE
				nStateAction := 80;
			END_IF
			fbStop(bExecute:= FALSE, DilSendCmd:= fbSendCmd);
		END_IF
		
END_CASE

//Errorhandling
IF nStateAction = 99 THEN
	stError.Cmd := E_Action.ACTION_DilMovePlunger;
	stError.POUAction := E_POUACT.POUACT_A_MovePlunger;
	fbErrorList.M_Add(stError);
END_IF
END_ACTION

ACTION A_MoveValve:
stError.POUState := nStateAction;

CASE nStateAction OF
	0:
		fbMoveValve(nValvePos:= nValvePosPump, bExecute:= TRUE, DilSendCmd:= fbSendCmd, pDilRef:= pDiluterRef1);
		
		IF NOT fbMoveValve.bBusy THEN
			IF fbMoveValve.bError THEN
				stError.ErrorId := fbMoveValve.nErrorId;
 				nStateAction := 99;
			ELSE
				//nCurValvePos := fbMoveValve.nCurrentPos;
				nStateAction := 80;
			END_IF
			fbMoveValve(bExecute:= FALSE, DilSendCmd:= fbSendCmd, pDilRef:= pDiluterRef1);
		END_IF
	
	70:	//Abbrechen
		fbMoveValve(bExecute:= FALSE, DilSendCmd:= fbSendCmd, pDilRef:= pDiluterRef1);
		nStateAction := 71;
		
	71:	
		fbStop(bExecute:= TRUE, DilSendCmd:= fbSendCmd, pDilRef1 := pDiluterRef1);
		
		IF NOT fbStop.bBusy THEN
			IF fbStop.bError THEN
				nStateAction := 99;
				stError.ErrorId := fbStop.nErrorId;
			ELSE
				nStateAction := 80;
			END_IF
			fbStop(bExecute:= FALSE, DilSendCmd:= fbSendCmd);
		END_IF		
END_CASE	

//Errorhandling
IF nStateAction = 99 THEN
	stError.Cmd := E_Action.ACTION_DilMoveValve;
	stError.POUAction := E_POUACT.POUACT_A_MoveValve;
	fbErrorList.M_Add(stError);
END_IF
END_ACTION

ACTION A_Prepare:
stError.POUState := nStateAction;

IF nStateAction = 0 THEN
	nStateAction := 1;
	IF ePrepareMode = E_DilPrepareMode.ForAspirate THEN
		//Abstand von ganz unten zu aktueller Pos muss mind TotalSteps betragen
		nSetPosPlunger := UDINT_TO_UINT(24000 - nTotalSteps);
		IF eReadedValveType = E_DilValveType.VALVETYPE_3Way THEN
			fbMoveToPos.nValvePos := nValvePosInput;
		ELSIF eReadedValveType = E_DilValveType.VALVETYPE_4Distribution THEN
			fbMoveToPos.nValvePos := nValvePosWaste;
		END_IF
		
		IF nSetPosPlunger >= pDiluterRef1^.nActPlungerPos THEN	//Kolbenposition breits passend
			//weiter zu MoveValve
			nStateAction := 2;
		END_IF
	ELSE //ForDispense
		nSetPosPlunger := UDINT_TO_UINT(nTotalSteps);
		fbMoveToPos.nValvePos := nValvePosInput;
		IF nSetPosPlunger <= pDiluterRef1^.nActPlungerPos THEN	//Kolbenposition bereits passend
			//weiter zu MoveValve
			nStateAction := 2;
		END_IF
	END_IF			
END_IF

IF nStateAction = 1 THEN	//Move plunger
	fbMoveToPos(bExecute:= TRUE, pDilRef:= pDiluterRef1, nTopSpeed:= DINT_TO_UINT(nSpeedReload), 
				nPosition:= nSetPosPlunger, DilSendCmd:= fbSendCmd);
	IF NOT fbMoveToPos.bBusy THEN
		IF fbMoveToPos.bError THEN
			stError.ErrorId := fbMoveToPos.nErrorId;
			nStateAction := 99;
		ELSE
			nStateAction := 2;
		END_IF
		fbMoveToPos(bExecute:= FALSE, pDilRef:= pDiluterRef1, DilSendCmd:= fbSendCmd);
	END_IF
END_IF

IF nStateAction = 2 THEN	//Move valve
	fbMoveValve(bExecute:= TRUE, nValvePos:= nValvePosOutput, pDilRef:= pDiluterRef1, DilSendCmd:= fbSendCmd);
	IF NOT fbMoveValve.bBusy THEN
		IF fbMoveValve.bError THEN
			stError.ErrorId := fbMoveValve.nErrorId;
			nStateAction := 99;
		ELSE
			nStateAction := 80;
		END_IF
		fbMoveValve(bExecute:= FALSE, pDilRef:= pDiluterRef1, DilSendCmd:= fbSendCmd);
	END_IF
END_IF

//Abbrechen
IF nStateAction = 70 THEN
	IF fbMoveToPos.bBusy THEN
		fbMoveToPos(bExecute:= FALSE, DilSendCmd:= fbSendCmd, pDilRef:= pDiluterRef1);
	ELSE
		nStateAction := 71;
	END_IF
END_IF

IF nStateAction = 71 THEN
	fbStop(bExecute:= TRUE, DilSendCmd:= fbSendCmd, pDilRef1 := pDiluterRef1);
	IF NOT fbStop.bBusy THEN
		IF fbStop.bError THEN
			nStateAction := 99;
			stError.ErrorId := fbStop.nErrorId;
		ELSE
			nStateAction := 80;
		END_IF
		fbStop(bExecute:= FALSE, DilSendCmd:= fbSendCmd);
	END_IF	
END_IF
//Ende Abbrechen

//Errorhandling
IF nStateAction = 99 THEN
	stError.Cmd := E_Action.ACTION_DilPrepare;
	stError.POUAction := E_POUACT.POUACT_A_Prepare;
	fbErrorList.M_Add(stError);
END_IF
END_ACTION

ACTION A_Pump:
stError.POUState := nStateAction;

IF nStateAction = 0 THEN
	//BottleStates abfragen
	stError.ErrorId := M_CheckBottles(0);
	IF stError.ErrorId > 0 THEN
		nStateAction := 70;
		nStateNext := 99;
		RETURN;
	END_IF	
	
	nStateNext := 80;
	fbPump(eMode:= ePumpMode, nValvePosPump:= nValvePosPump, nValvePosReload:= nValvePosReload, 
			nSpeedPump:= nSpeedPump, nSpeedReload:= nSpeedReload, nTotalSteps:= nTotalSteps,
			bExecute:= TRUE, DilSendCmd:= fbSendCmd, pDilRef:= pDiluterRef1, bEndless:= bEndless, bFirstReload:= bFirstReload);
	IF NOT fbPump.bBusy THEN
		IF fbPump.bError THEN
			bError := TRUE;
			stError.ErrorId := fbPump.nErrorId;
			nStateAction := 99;
		ELSE
			nStateAction := 80;				
		END_IF
		fbPump(bExecute:= FALSE, DilSendCmd:= fbSendCmd, pDilRef:= pDiluterRef1);
	END_IF
END_IF

//Abbrechen
IF nStateAction = 70 THEN
	IF fbPump.bBusy THEN
		fbPump(bExecute:= FALSE, DilSendCmd:= fbSendCmd, pDilRef:= pDiluterRef1);
	ELSE
		nStateAction := 71;
	END_IF
END_IF

IF nStateAction = 71 THEN
	fbStop(bExecute:= TRUE, DilSendCmd:= fbSendCmd, pDilRef1 := pDiluterRef1);
	IF NOT fbStop.bBusy THEN
		IF fbStop.bError THEN
			nStateAction := 99;
			stError.ErrorId := fbStop.nErrorId;
		ELSE
			nStateAction := nStateNext;
		END_IF
		fbStop(bExecute:= FALSE, DilSendCmd:= fbSendCmd);
	END_IF	
END_IF
//Ende Abbrechen

//Errorhandling
IF nStateAction = 99 THEN
	fbPump(bExecute:= FALSE, DilSendCmd:= fbSendCmd, pDilRef:= pDiluterRef1);
	stError.Cmd := E_Action.ACTION_DilPump;
	stError.POUAction := E_POUACT.POUACT_A_Pump;
	fbErrorList.M_Add(stError);
END_IF
END_ACTION

ACTION A_Reset:
CASE nStateA_Reset OF
	0:
		nStateA_Reset := 80;
END_CASE
END_ACTION

ACTION A_Stop:
IF nStateA_Stop = 0 THEN
	//Init lässt sich beim Diluter nicht abbrechen
	IF bMovePlunger AND nStateAction < 70 THEN
		nStateAction := 70;
	END_IF

	IF bMoveValve AND nStateAction < 70 THEN
		nStateAction := 70;
	END_IF

	IF bPump AND nStateAction < 70 THEN
		nStateAction := 70;
	END_IF
	
	IF bTransfer AND nStateAction < 70 THEN
		nStateAction := 70;
	END_IF
	
	IF bPrepare AND nStateAction = 1 THEN
		nStateAction := 70;
	END_IF
	
 	nStateA_Stop := 1;
	
ELSIF nStateA_Stop = 1 THEN	//Warten bis Action abgebrochen
	IF NOT (bInit OR bMovePlunger OR bMoveValve OR bPump OR bTransfer OR bPrepare) THEN
		nStateA_Stop := 80;
	END_IF
END_IF
END_ACTION

ACTION A_Transfer:
stError.POUState := nStateAction;

IF nStateAction = 0 THEN
	//BottleStates abfragen
	stError.ErrorId := M_CheckBottles(0);
	IF stError.ErrorId > 0 THEN
		nStateAction := 70;
		nStateNext := 99;
		RETURN;
	END_IF
	
	stError.ErrorId := pDilRefDest^.M_CheckBottles(0);
	IF stError.ErrorId > 0 THEN
		nStateAction := 70;
		nStateNext := 99;
		RETURN;
	END_IF
	
	nStateNext := 80;
	fbTransfer(nTransferSteps:= nTotalSteps,
				nPreSteps:= nPreSteps, nPostSteps:= nPostSteps,
				nValveInput1:= nValvePosInput,
				nValveOutput1:= nValvePosOutput,
				nValveWaste1:= nValvePosWaste,
				nValveInput2:= pDilRefDest^.P_nValvePosInput,
				nValveOutput2:= pDilRefDest^.P_nValvePosOutput,
				nValveWaste2:= pDilRefDest^.P_nValvePosWaste,
				nSpeedPump:= nSpeedPump, nSpeedReload:= nSpeedReload, bExecute:= TRUE,
				DilSendCmd:= fbSendCmd, pDilRef1:= pDiluterRef1, pDilRef2:= pDilRefDest^.P_pDilRef);

	IF NOT fbTransfer.bBusy THEN
		IF fbTransfer.bError THEN
			bError := TRUE;
			stError.ErrorId := fbTransfer.nErrorId;
			nStateAction := 99;
		ELSE
			fbTransfer(bExecute:= FALSE, DilSendCmd:= fbSendCmd);
			nStateAction := 80;				
		END_IF
		fbTransfer(bExecute:= FALSE, DilSendCmd:= fbSendCmd);
	END_IF
END_IF
	
//Abbrechen
IF nStateAction = 70 THEN
	IF fbTransfer.bBusy THEN
		fbTransfer(bExecute:= FALSE, DilSendCmd:= fbSendCmd);
	ELSE
		nStateAction := 71;
	END_IF
END_IF
		
IF nStateAction = 71 THEN //Dil1+Dil2 stoppen 
	fbStop(bExecute:= TRUE, DilSendCmd:= fbSendCmd, pDilRef1:= pDiluterRef1, pDilRef2:= pDilRefDest^.P_pDilRef);
	IF NOT fbStop.bBusy THEN
		IF fbStop.bError THEN
			nStateAction := 99;
			stError.ErrorId := fbStop.nErrorId;
		ELSE
			nStateAction := 80;
		END_IF
		fbStop(bExecute:= FALSE, DilSendCmd:= fbSendCmd);
	END_IF
END_IF
		
//Ende Abbrechen

//Errorhandling
IF nStateAction = 99 THEN
	stError.Cmd := E_Action.ACTION_DilTransfer;
	stError.POUAction := E_POUACT.POUACT_A_TransferLiquid;
	fbErrorList.M_Add(stError);
END_IF
END_ACTION

METHOD FB_init : BOOL
VAR_INPUT
	bInitRetains : BOOL; // if TRUE, the retain variables are initialized (warm start / cold start)
	bInCopyCode : BOOL;  // if TRUE, the instance afterwards gets moved into the copy code (online change)
END_VAR
eObjectType := E_ObjectType.OBJECTTYPE_Diluter;
eObjectGroup := E_ObjectGroup.OBJECTGROUP_Device;
END_METHOD

METHOD M_CancelAction
VAR_INPUT
	eAction : E_Action;
END_VAR
CASE eAction OF
	E_Action.ACTION_DilMovePlunger:
		IF bMovePlunger AND nStateAction < 70 THEN
			nStateAction := 70;
		END_IF	
	E_Action.ACTION_DilMoveValve:
		IF bMoveValve AND nStateAction < 70 THEN
			nStateAction := 70;
		END_IF	
	E_Action.ACTION_DilPump:
		IF bPump AND nStateAction < 70 THEN
			nStateAction := 70;
		END_IF	
	E_Action.ACTION_DilTransfer:
		IF bTransfer AND nStateAction < 70 THEN
			nStateAction := 70;
		END_IF
	E_Action.ACTION_DilPrepare:
		IF bPrepare AND nStateAction = 1 THEN
			nStateAction := 70;
		END_IF
END_CASE
END_METHOD

METHOD M_CheckAction : ERRORID
VAR_INPUT
	refActionData 	: REFERENCE TO ST_ActionData;
	pCorrelObject	: POINTER TO FB_Object;
END_VAR
M_CheckAction := E_ErrorIdCmd.ERRORID_InvalidAction;
END_METHOD

METHOD M_CheckBottles : ERRORID
VAR_INPUT
	nInputNr : USINT; //wird nur bei FB_Diluter3Inputs genutzt
END_VAR
//Systemliquidbottle OK?
IF nSysLiquidBottle > 0 THEN
	IF NOT aSensSysLiquidBottle[nSysLiquidBottle] THEN //Leer
		M_CheckBottles := E_ErrorIdCmd.ERRORID_LiquidBottleEmpty;
		RETURN;
	END_IF
END_IF
//Wastebottle OK?
IF nWasteBottle > 0 THEN
	IF NOT aSensWasteBottle[nWasteBottle] THEN //Voll
		M_CheckBottles := E_ErrorIdCmd.ERRORID_WasteBottleFull;
		RETURN;
	END_IF
END_IF
END_METHOD

METHOD M_CheckProcDataType : BOOL
VAR_INPUT
	eProcDataType : E_ProcDataType;
END_VAR
END_METHOD

METHOD M_CheckProps : ERRORID
VAR_INPUT
END_VAR
//richtige Spritzgröße konfiguriert?
IF NOT (nSyringeSize = 50 OR nSyringeSize = 100 OR nSyringeSize = 250 OR nSyringeSize = 500 OR nSyringeSize = 1000 OR nSyringeSize = 2500 OR nSyringeSize = 5000) THEN
	M_CheckProps := E_ErrorIdDiluter.ERRORID_InvalidSyringe; //Falsche Spritzgröße konfiguriert - Error
END_IF
END_METHOD

METHOD M_CheckSpeed : ERRORID
VAR_INPUT
	nValue : DINT;
END_VAR
IF (nValue < 5) THEN	//minimale Geschwindigkeit darf 5 Halbsteps/s nicht unterschreiten
	M_CheckSpeed := E_ErrorIdDiluter.ERRORID_SpeedToSmall;
ELSIF (nValue > 5200) THEN	//maximale Geschwindigkeit darf 5200 Halbsteps/s nicht überschreiten
	M_CheckSpeed := E_ErrorIdDiluter.ERRORID_SpeedExeeded;
END_IF
END_METHOD

METHOD M_ClearAllProps
VAR_INPUT
	bIgnoreParent : BOOL; //Es wird das gesamte OD gelöscht. -> Zeiger auf Parent nicht mehr gültig!
END_VAR
SUPER^.M_ClearAllProps(bIgnoreParent);
pDiluterRef1 := 0;
END_METHOD

METHOD M_ExeAction : ERRORID
VAR_INPUT
	refActionData	: REFERENCE TO ST_ActionData;
END_VAR

VAR
	sTemp : STRING(2);
	nTransferDestDil : UINT;
END_VAR
//Diluter kann keine Actions parallel ausführen
//Die einzige Action ist Stop
IF eCurrentState = E_MachineState.MACHINESTATE_Idle THEN
	CASE refActionData.eAction OF
		E_Action.ACTION_Init:	//Diluter initialisieren
			IF NOT bInit THEN
				bInit := TRUE;
				bReInit := DINT_TO_BOOL(refActionData.aParams[1]);
			ELSE
				RETURN;
			END_IF
			
		E_Action.ACTION_DilMovePlunger:
			IF NOT bIsInit THEN
				M_ExeAction := E_ErrorIdDiluter.ERRORID_NotIniialized;
				RETURN;
			END_IF
			nSetPosPlunger := DINT_TO_UINT(refActionData.aParams[1]);
			IF nSetPosPlunger < 0 OR nSetPosPlunger > 24000 THEN
				M_ExeAction := E_ErrorIdDiluter.ERRORID_InvalidPlungerPos;  //Error
				RETURN;
			END_IF
			//Flow von 10tel µl/s in Halbsteps/s umrechnen (1 voller Hub sind 6000 Halbsteps)
			//Die minimale Geschwindigkeit darf 5 Halbsteps/s nicht unterschreiten
			//nSpeedPump := (refActionData.aParams[2] * 6000) /10 / nSyringeSize;
			nSpeedPump := F_DilFlowToSpeed(refActionData.aParams[2], nSyringeSize);
			IF nSpeedPump > 5200 THEN	//Error
				M_ExeAction := E_ErrorIdDiluter.ERRORID_SpeedExeeded;
				RETURN;
			END_IF			
			nValvePosPump := DINT_TO_SINT(refActionData.aParams[3]);
			bMovePlunger := TRUE;
	
		E_Action.ACTION_DilMoveValve:
			IF NOT bIsInit THEN
				M_ExeAction := E_ErrorIdDiluter.ERRORID_NotIniialized;
				RETURN;
			END_IF
			nValvePosPump := DINT_TO_SINT(refActionData.aParams[1]);
			bMoveValve := TRUE;
			
		E_Action.ACTION_DilPump: //Diluter Pumpen
			IF NOT bIsInit THEN
				M_ExeAction := E_ErrorIdDiluter.ERRORID_NotIniialized;
				RETURN;
			END_IF
			//Param1 = Quantity in 10tel µl
			//Param2 = Mode (Saugen oder Drücken)
			//Param3 = Flow Pumpen in 10tel µl/sec
			//Param4 = Flow Nachladen in 10tel µl/sec
			//Param5 = Ventilstellung Pump
			//Param6 = Ventilstellung Nachladen
			//Param7 = endless
			//Param8 = firstReload 
			
			//Bottles OK?
			M_ExeAction := M_CheckBottles(0);
			IF M_ExeAction > 0 THEN
				RETURN;
			END_IF
	
			ePumpMode := DINT_TO_USINT(refActionData.aParams[1]);
			
			//Umrechnung von 10tel µl in Mircosteps
			nTotalSteps := F_DilQuantityToMicroSteps(refActionData.aParams[2],nSyringeSize);
			
			//Umrechnung 10tel µl/s in Halbsteps/s
			nSpeedPump := F_DilFlowToSpeed(refActionData.aParams[3], nSyringeSize);
	
			M_ExeAction := M_CheckSpeed(nSpeedPump);
			IF M_ExeAction > 0 THEN
				RETURN;
			END_IF
			
			IF refActionData.aParams[4] = 0 THEN
				//Umrechnung 10tel µl/s in Halbsteps/s
				nSpeedReload := F_DilFlowToSpeed(nConfigReloadSpeed, nSyringeSize);
			ELSE
				//Umrechnung 10tel µl/s in Halbsteps/s
				nSpeedReload := F_DilFlowToSpeed(refActionData.aParams[4], nSyringeSize);
			END_IF
			M_ExeAction := M_CheckSpeed(nSpeedReload);
			IF M_ExeAction > 0 THEN
				RETURN;
			END_IF			
			//Valve-Position Pumpen ermitteln
			IF refActionData.aParams[5] = 0 THEN
				nValvePosPump := nValvePosOutput;
			ELSE
				nValvePosPump := DINT_TO_SINT(refActionData.aParams[5]);
			END_IF
			//Valve-Position Reload ermitteln
			IF refActionData.aParams[6] = 0 THEN
				IF ePumpMode = E_DilPumpMode.MODE_Press THEN
					nValvePosReload := nValvePosInput;
				ELSE //Suck
					IF eReadedValveType = E_DilValveType.VALVETYPE_3Way THEN
						nValvePosReload := nValvePosInput;
					ELSIF eReadedValveType = E_DilValveType.VALVETYPE_4Distribution THEN
						nValvePosReload := nValvePosWaste;
					END_IF
				END_IF
			ELSE
				nValvePosReload := DINT_TO_SINT(refActionData.aParams[6]);
			END_IF
			bEndless := DINT_TO_BOOL(refActionData.aParams[7]);
			bFirstReload := DINT_TO_BOOL(refActionData.aParams[8]);
			bPump := TRUE;
			
		E_Action.ACTION_DilTransfer:
			IF NOT bIsInit THEN
				M_ExeAction := E_ErrorIdDiluter.ERRORID_NotIniialized;
				RETURN;
			END_IF
				//Diluter Destination ermitteln
			nTransferDestDil := DINT_TO_UINT(refActionData.aParams[1]);
			IF fbObjectDirectory.M_GetObjType(nTransferDestDil) = E_ObjectType.OBJECTTYPE_Diluter THEN
				pDilRefDest := fbObjectDirectory.M_GetObjPointer(nTransferDestDil);
			ELSE
				M_ExeAction:= E_ErrorIdCmd.ERRORID_UnsuitableObject;
				RETURN;
			END_IF
			
			//Bottles DilSrc OK?
			M_ExeAction := M_CheckBottles(0);
			IF M_ExeAction > 0 THEN
				RETURN;
			END_IF
	
			//Bottles DilDest OK?
			M_ExeAction := pDilRefDest^.M_CheckBottles(0);
			IF M_ExeAction > 0 THEN
				RETURN;
			END_IF
			
			//Menge von 10tel µl in Microsteps umrechnen
			nTotalSteps := F_DilQuantityToMicroSteps(refActionData.aParams[2],nSyringeSize);
	
			//Umrechnung 10tel µl/s in Halbsteps/s
			nSpeedPump := F_DilFlowToSpeed(refActionData.aParams[3], nSyringeSize);
			
			M_ExeAction := M_CheckSpeed(nSpeedPump);
			IF M_ExeAction > 0 THEN
				RETURN;
			END_IF
			
			//Umrechnung 10tel µl/s in Halbsteps/s
			nSpeedReload := F_DilFlowToSpeed(nConfigReloadSpeed, nSyringeSize);
			
			M_ExeAction := M_CheckSpeed(nSpeedReload);
			IF M_ExeAction > 0 THEN
				RETURN;
			END_IF
			nPreSteps := UDINT_TO_INT(F_DilQuantityToMicroSteps(refActionData.aParams[4],nSyringeSize));
			nPostSteps := UDINT_TO_INT(F_DilQuantityToMicroSteps(refActionData.aParams[5],nSyringeSize));
			bTransfer := TRUE;
			
		E_Action.ACTION_DilPrepare:
			IF NOT bIsInit THEN
				M_ExeAction := E_ErrorIdDiluter.ERRORID_NotIniialized;
				RETURN;
			END_IF
			//Bottles OK?
			M_ExeAction := M_CheckBottles(0);
			IF M_ExeAction > 0 THEN
				RETURN;
			END_IF
			
			ePrepareMode := DINT_TO_USINT(refActionData.aParams[1]);
			//Umrechnung von 10tel µl in Mircosteps
			nTotalSteps := F_DilQuantityToMicroSteps(refActionData.aParams[2],nSyringeSize);
			nTotalSteps := MIN(24000,nTotalSteps);	//Es kann für max einen Hub reloaded werden
			nSpeedReload := F_DilFlowToSpeed(nConfigReloadSpeed, nSyringeSize);
			bPrepare := TRUE;
		E_Action.ACTION_Stop:
			//do nothing
		ELSE
			M_ExeAction := E_ErrorIdCmd.ERRORID_InvalidAction;
	END_CASE
	bBusy := TRUE;
	eCurrentAction := refActionData.eAction;
	eCurrentState := E_MachineState.MACHINESTATE_Active;
ELSIF (eCurrentState = E_MachineState.MACHINESTATE_Active) AND (refActionData.eAction = E_Action.ACTION_Stop) THEN
	M_Stop();
ELSE
	M_ExeAction := E_ErrorIdCmd.ERRORID_InvalidState;
	RETURN;
END_IF
END_METHOD

METHOD M_GetActionBusy : BOOL
VAR_INPUT
	eAction : E_Action;
END_VAR
IF eAction = eCurrentAction THEN
	M_GetActionBusy := TRUE;	
END_IF
END_METHOD

METHOD M_GetAllProps : ERRORID
VAR_INPUT
	refCmdData : REFERENCE TO  ST_CmdData;
END_VAR
refCmdData.aHeader[0] := nObjectID;
refCmdData.aHeader[1] := eObjectType;
refCmdData.aHeader[2]:= nNotifyId;

refCmdData.n32Data[1] := nParentSlotNr;
refCmdData.n32Data[2] := nChannel;		//Diluter-Kanal
refCmdData.n32Data[3] := nSyringeSize;	//Spritzengröße (für beide Dilutoren)
refCmdData.n32Data[4] := nSysLiquidBottle;
refCmdData.n32Data[5] := nWasteBottle;
refCmdData.n32Data[6] := nConfigReloadSpeed;
refCmdData.n32Data[7] := eValveType;
refCmdData.n32Data[8] := nValvePosInput;
refCmdData.n32Data[9] := nValvePosOutput;
refCmdData.n32Data[10] := nValvePosWaste;
END_METHOD

METHOD M_GetDevice : I_Device
VAR_INPUT
END_VAR
M_GetDevice := THIS^;
END_METHOD

METHOD M_GetProcData : DINT
VAR_INPUT
	eProcDataType : E_ProcDataType;
END_VAR
END_METHOD

METHOD M_Reset
bBusy := TRUE;
eCurrentState := E_MachineState.MACHINESTATE_Reset;
END_METHOD

METHOD M_SetAllProps : ERRORID
VAR_INPUT
	refCmdData : REFERENCE TO  ST_CmdData;
END_VAR
nNoOfProps := 11;

nParentSlotNr := DINT_TO_UINT(refCmdData.n32Data[1]);

//Diluterkanal checken
//Channel muss zwischen 1 und 7 liegen
IF  NOT((refCmdData.n32Data[2] > 0) AND (refCmdData.n32Data[2] <= cNoOfDiluters)) THEN
	M_SetAllProps := E_ErrorIdObjMgmt.ERRORID_InvalidDiluterChannel;
	RETURN;
ELSE
	nChannel := DINT_TO_USINT(refCmdData.n32Data[2]);
	pDiluterRef1 := ADR(aFbDiluterRef[nChannel]);
END_IF

//Spritzengröße
IF NOT (refCmdData.n32Data[3] = 50 OR 
		refCmdData.n32Data[3] = 100 OR 
		refCmdData.n32Data[3] = 250 OR 
		refCmdData.n32Data[3] = 500 OR 
		refCmdData.n32Data[3] = 1000 OR
		refCmdData.n32Data[3] = 2500 OR
		refCmdData.n32Data[3] = 5000) THEN
		M_SetAllProps := E_ErrorIdObjMgmt.ERRORID_InvalidSyringeSize;
ELSE
	nSyringeSize := refCmdData.n32Data[3];
END_IF

//Systemliquidbottle Dil
IF refCmdData.n32Data[4] >= 0 AND refCmdData.n32Data[4] <= cNoOfLiquidBottles THEN
	nSysLiquidBottle := DINT_TO_USINT(refCmdData.n32Data[4]);
ELSE
	M_SetAllProps := E_ErrorIdObjMgmt.ERRORID_InvalidLiquidbottle;
	RETURN;
END_IF

//Wastebottle Dil
IF refCmdData.n32Data[5] >= 0 AND refCmdData.n32Data[5] <= cNoOfWasteBottles THEN
	nWasteBottle := DINT_TO_USINT(refCmdData.n32Data[5]);
ELSE
	M_SetAllProps := E_ErrorIdObjMgmt.ERRORID_InvalidWastebottle;
	RETURN;
END_IF

//ReloadSpeed
nConfigReloadSpeed := refCmdData.n32Data[6];

//ValveType
eValveType := DINT_TO_USINT(refCmdData.n32Data[7]);
IF NOT(eValveType = E_DilValveType.VALVETYPE_3Way OR eValveType = E_DilValveType.VALVETYPE_4Distribution) THEN
	M_SetAllProps := E_ErrorIdDiluter.ERRORID_InvalidValveType;
	RETURN;
END_IF

nValvePosInput := DINT_TO_SINT(refCmdData.n32Data[8]);
nValvePosOutput := DINT_TO_SINT(refCmdData.n32Data[9]);
nValvePosWaste := DINT_TO_SINT(refCmdData.n32Data[10]);
END_METHOD

METHOD M_SetSingleProp : ERRORID
VAR_INPUT
	refCmdData : REFERENCE TO  ST_CmdData;
END_VAR
//Diluter besitzt nur Specialproperties
CASE refCmdData.aHeader[1] OF	//Property-Nr
	2:	//Channel muss zwischen 1 und 7 liegen
		IF  NOT((refCmdData.n32Data[0] > 0) AND (refCmdData.n32Data[0] <= cNoOfDiluters)) THEN
			M_SetSingleProp := E_ErrorIdObjMgmt.ERRORID_InvalidDiluterChannel;
			RETURN;
		ELSE
			nChannel := DINT_TO_USINT(refCmdData.n32Data[0]);
			pDiluterRef1 := ADR(aFbDiluterRef[nChannel]);
		END_IF	
		
	3:	//SyringeSize	
		IF NOT (refCmdData.n32Data[0] = 50 OR 
				refCmdData.n32Data[0] = 100 OR 
				refCmdData.n32Data[0] = 250 OR 
				refCmdData.n32Data[0] = 500 OR 
				refCmdData.n32Data[0] = 1000 OR 
				refCmdData.n32Data[0] = 5000) THEN
				M_SetSingleProp := E_ErrorIdObjMgmt.ERRORID_InvalidSyringeSize;
		ELSE
			nSyringeSize := refCmdData.n32Data[0];
		END_IF

	4:	//Systemliquidbottle
		IF refCmdData.n32Data[0] >= 0 AND refCmdData.n32Data[0] <= cNoOfLiquidBottles THEN
			nSysLiquidBottle := DINT_TO_USINT(refCmdData.n32Data[0]);
		ELSE
			M_SetSingleProp := E_ErrorIdObjMgmt.ERRORID_InvalidLiquidbottle;
		END_IF		
	5:	//Wastebottle
		IF refCmdData.n32Data[0] >= 0 AND refCmdData.n32Data[0] <= cNoOfWasteBottles THEN
			nWasteBottle := DINT_TO_USINT(refCmdData.n32Data[0]);
		ELSE
			M_SetSingleProp := E_ErrorIdObjMgmt.ERRORID_InvalidWastebottle;
		END_IF		

	6:	//RelaodSpeed
		nConfigReloadSpeed := refCmdData.n32Data[0];
		
	8:	//ValvePosInput
		nValvePosInput := DINT_TO_SINT(refCmdData.n32Data[0]);
		
	9:	//ValvePosOutput
		nValvePosOutput := DINT_TO_SINT(refCmdData.n32Data[0]);
		
	10:	//ValvePosWaste
		nValvePosWaste := DINT_TO_SINT(refCmdData.n32Data[0]);

	ELSE
		//Ungültige Property-Nr
		M_SetSingleProp := E_ErrorIdCmd.ERRORID_InvalidProperty;
END_CASE
END_METHOD

METHOD M_Stop : ERRORID
VAR_INPUT
END_VAR
VAR
	
END_VAR
IF bBusy THEN
	bStop := TRUE;	
END_IF
END_METHOD

PROPERTY P_bBusy : BOOL
GET
P_bBusy := bBusy;
END_GET
END_PROPERTY

PROPERTY P_bCanceled : BOOL
GET
P_bCanceled := bCanceled;
END_GET
END_PROPERTY

PROPERTY P_bError : BOOL
GET
IF eCurrentState = E_MachineState.MACHINESTATE_Error THEN
	P_bError := TRUE;
END_IF
END_GET
END_PROPERTY

PROPERTY P_bIsInit : BOOL
GET
P_bIsInit := bIsInit;
END_GET
SET
bIsInit := P_bIsInit;
END_SET
END_PROPERTY

PROPERTY P_bStopAllOnError : BOOL
GET
P_bStopAllOnError := bStopAllOnError;
END_GET
END_PROPERTY

PROPERTY P_eCurrentState : E_MachineState
GET
P_eCurrentState := eCurrentState;
END_GET
END_PROPERTY

PROPERTY P_nConfigReloadSpeed : DINT
GET
P_nConfigReloadSpeed := nConfigReloadSpeed;
END_GET
END_PROPERTY

PROPERTY P_nCurValvePos : SINT
GET
IF pDiluterRef1 > 0 THEN
	P_nCurValvePos := pDiluterRef1^.nActValvePos;
END_IF
END_GET
END_PROPERTY

PROPERTY P_nErrorId : ERRORID
GET
P_nErrorID := nErrorID;
END_GET
END_PROPERTY

PROPERTY P_nNotifyId : UINT
GET
P_nNotifyId := nNotifyId;
END_GET
SET
nNotifyId := P_nNotifyId;
END_SET
END_PROPERTY

PROPERTY P_nParentSlotNr : UINT
GET
P_nParentSlotNr := nParentSlotNr;
END_GET
END_PROPERTY

PROPERTY P_nSyringeSize : DINT
GET
P_nSyringeSize := nSyringeSize;
END_GET
END_PROPERTY

PROPERTY P_nValvePosInput : SINT
GET
P_nValvePosInput := nValvePosInput;
END_GET
END_PROPERTY

PROPERTY P_nValvePosOutput : SINT
GET
P_nValvePosOutput := nValvePosOutput;
END_GET
END_PROPERTY

PROPERTY P_nValvePosWaste : SINT
GET
P_nValvePosWaste := nValvePosWaste;
END_GET
END_PROPERTY

PROPERTY P_pDilRef : POINTER TO FB_HwRefDiluter
GET
P_pDilRef := pDiluterRef1;
END_GET
END_PROPERTY

PROPERTY P_pObject : POINTER TO FB_Object
GET
P_pObject := THIS;
END_GET
END_PROPERTY

PROPERTY P_stError : ST_Error
GET
P_stError := stError;
END_GET
END_PROPERTY

END_FUNCTION_BLOCK

// ---- Hardware/Diluter/FB_HwRefDiluter.TcPOU
FUNCTION_BLOCK FB_HwRefDiluter
VAR_INPUT
	bIsInit 		: BOOL;
	bBusy			: BOOL;
	eValveType 		: E_DilValveType;
	nActValvePos	: SINT;
	nActPlungerPos	: UINT;	
END_VAR
VAR_OUTPUT
	nChannel		: USINT;
END_VAR
VAR
END_VAR
VAR_STAT
	nHighestChannel : USINT;
END_VAR

METHOD FB_init : BOOL
VAR_INPUT
	bInitRetains : BOOL; // if TRUE, the retain variables are initialized (warm start / cold start)
	bInCopyCode : BOOL;  // if TRUE, the instance afterwards gets moved into the copy code (online change)
END_VAR
nHighestChannel := nHighestChannel + 1;
nChannel := nHighestChannel;
END_METHOD

END_FUNCTION_BLOCK

// ---- Hardware/Diluter/FB_Dil_GetPlungerPos.TcPOU
FUNCTION_BLOCK FB_Dil_GetPlungerPos
VAR_INPUT
	bExecute	: BOOL;
	pDilRef		: POINTER TO FB_HwRefDiluter;
END_VAR
VAR_OUTPUT
	bBusy		: BOOL;
	bError		: BOOL;
	nErrorId	: ERRORID;
	nValue		: UINT;
	bStatus		: BOOL;
END_VAR
VAR
	rTrig : R_TRIG;
	pDilRefIntern : POINTER TO FB_HwRefDiluter;
END_VAR
VAR_IN_OUT
	DilSendCmd 	: FB_Dil_SendCmd;
END_VAR

rTrig(CLK:= bExecute);
IF rTrig.Q THEN
	IF pDilRef = 0 THEN
		bError := TRUE;
		RETURN;	
	ELSE
		pDilRefIntern := pDilRef;
	END_IF	
END_IF

IF bExecute THEN
	bBusy := TRUE;

	DilSendCmd(bExecute:= TRUE, bExpectReply:= TRUE, sSendData:= CONCAT(USINT_TO_STRING(pDilRefIntern^.nChannel),'?0'));
	
	IF NOT DilSendCmd.bBusy THEN
		IF DilSendCmd.bError THEN
			bError := TRUE;
			nErrorId := DilSendCmd.nErrorId;
		ELSE
			IF DilSendCmd.bDataIsNumeric THEN
				nValue := STRING_TO_UINT(DilSendCmd.sReceiveData);
				pDilRefIntern^.nActPlungerPos := nValue; 
			END_IF
			bStatus := DilSendCmd.bStatus;
		END_IF
		DilSendCmd(bExecute:= FALSE);
		bBusy := FALSE;
	END_IF
ELSE
	bBusy := FALSE;
	bError := FALSE;
	nErrorId := 0;
	nValue := 0;
	bStatus := FALSE;
END_IF

END_FUNCTION_BLOCK

// ---- Hardware/Diluter/FB_Dil_SendCmd.TcPOU
FUNCTION_BLOCK FB_Dil_SendCmd
VAR_INPUT
	bExecute		: BOOL;	
	bExpectReply	: BOOL; //Antwort vom Diluter wird erwartet
	sSendData		: STRING(100); //CommandString ohne CheckSum und Steuerzeichen	
END_VAR
VAR_OUTPUT
	bBusy			: BOOL;
	bError			: BOOL;
	nErrorId		: ERRORID; 	//RS232-Fehler oder vom Diluter zurückgegebener Fehler
	bStatus			: BOOL;		//Statusbit in Diluterantwort(True = device is ready for new commands)
	sReceiveData	: STRING;	//Datenstring bei zurückgegebenen Daten
	bDataIsNumeric	: BOOL; 	//True, wenn "sReceiveData" nur aus Zahlen besteht	
END_VAR
VAR_IN_OUT
	
END_VAR
VAR
	nState			: USINT;
	fbSendData		: Tc2_SerialCom.SendData;
	fbReceiveByte	: Tc2_SerialCom.ReceiveByte;
	fbReceiveData	: Tc2_SerialCom.ReceiveData;
	SerialPort		: REFERENCE TO FB_SerialComPort_Base;
	
	nPrefix			: BYTE := 2; //STX
	nSuffix			: BYTE := 3; //ETX
	timer1			: TON; 	//Timeout
	bFlag			: BOOL := TRUE;
	
	sSendString		: STRING(100); //temporärer Sendestring, welcher bis bis zur Checksumme exitstiert(danach in ByteArray)
	aSendData		: ARRAY[1..100] OF BYTE; //ByteArray, welches den kompletten SendeString incl. CheckSum aufnimmt
	aReceiveData	: ARRAY[0..30] OF BYTE; //ByteArray, welcher den EmpfangsString enthält (zwischen bzw. incl. STX und ETX)
	nLenData		: USINT; //komplette Länge der Sende-oder Empfamgsdaten
	nLenDatablock	: USINT; //Länge der empfangenen Datablocks (Positionen oder ausgelesene Parameter usw)
	nCheckSum		: BYTE; //Checksumme
	sChar			: STRING(2);
	i				: USINT;	
END_VAR

IF bExecute THEN
	IF nState = 0 THEN
		IF NOT __ISVALIDREF(SerialPort) THEN
			bError := TRUE;
			RETURN;
		END_IF
		//Am Serial Port zu Senden registrieren
		//Die Registrierung sollte, wenn alles richtig programmiert wurde, immer klappen!
		IF NOT SerialPort.M_Register(THIS) THEN
			bError := TRUE;
			RETURN;
		ELSE
			nState := 1	;
		END_IF
		bBusy := TRUE;
		bDataIsNumeric := FALSE;
	END_IF
	
	//Checken, ob an der Reihe (wird übersprungen, wenn "SerialPort.M_Register" TRUE zurückgibt
	IF nState = 1 THEN
		IF SerialPort.M_IsMyTurn(THIS) THEN
			nState := 2;
		END_IF
	END_IF
	
	//Ist an der Reihe
	IF nState = 2 THEN
		//Kommunikationspuffer löschen (nicht der Hardware-Buffer)
		SerialPort.M_ClearTxComBuffer();
		SerialPort.M_ClearRxComBuffer();
		
		//# # # # # # # # # # # # # Sendestring zusammensetzen # # # # # # # # # # # # # # # # # # #
		
		//die DeviceNr befindet sich bereits in "sSendString" -> STX davor setzen!!
		sSendString := CONCAT(CHR(2),sSendData);
		//an dritte Stelle die Sequenznummer 1 einfügen
		sSendString := INSERT(sSendString,'1',2);	
		//am Ende ETX anhängen
		sSendString := CONCAT(sSendString,CHR(3));
		//Checksumme aus bisherigem String bilden
		nCheckSum := F_GetCheckSumFromString(sSendString);
		
		//Die Checksumme kann nicht direkt an den String angehängt werden, da für den Fall, dass die Checksumme 0 ist,
		//das ASCII-Zeichen "NUL" entsteht, und dieses bei Strings als Terminierung gilt.
		//Der bisherige String muss also in ein Bytearray übertragen werden und die Checksumme wird dort als letztes angehängt.
		//Gesendet wird dann über "SendData" und nicht mehr mit SendString!!!
		
		//Bisherigen String in Byterarray schieben
		FOR i:= 1 TO INT_TO_USINT(LEN(sSendString)) BY 1 DO
			aSendData[i]:= ASC(MID(STR:= sSendString, LEN:= 1, POS:= i));
		END_FOR
		
		//CheckSum anhängen
		nLenData := i;
		aSendData[i]:= nCheckSum;
		
		nState := 3;	//weiter zu String senden
	END_IF
	
	CASE nState OF
		3:	//# # # # # # # # # # # # # Daten senden # # # # # # # # # # # # # # # # # # #
			IF bFlag XOR fbSendData.Busy THEN
				bFlag := FALSE;
				fbSendData(pSendData:= ADR(aSendData),Length:= nLenData, TXbuffer:= SerialPort.P_TxBuffer);
			END_IF
			
			IF NOT fbSendData.Busy THEN	//Sendung abgeschlossen
				IF fbSendData.Error > 0 THEN
					nErrorId := INT_TO_UINT(fbSendData.Error);
					bError := TRUE;
					bBusy := FALSE;
					nState := 99;
					RETURN;				
				ELSE
					IF bExpectReply THEN	//Antwort wird erwartet
						//10ms auf Antwort warten DAS KANN ZUR NOT ENTFALLEN?
						timer1(IN:= TRUE,PT:= T#20MS);
						IF timer1.Q THEN
							timer1(IN:= FALSE);
							nState := 4;	//weiter zu Daten empfangen
						END_IF;
					ELSE	//Antwort wird nicht erwartet -> Daten nicht abrufen
						bBusy := FALSE;
						nState:= 80;	//FB ready	
					END_IF
				END_IF
			END_IF
		
		4:	//# # # # # # # # # # # # # Daten empfangen # # # # # # # # # # # # # # # # # # #
			//wenn keine Antwort erwartet wird (z.B. Command an mehrere Diluter gleichzeitig,
			// dann diesen Schritt überspringen, da sonst ein Timeout eintritt
			//wenn inerhalb von 200ms nicht emfangen  wurde, dann in Timeout-Fehler gehen
			
			timer1(IN:= TRUE,PT:= T#200MS);	//Timer für Timeout starten
			//In dieser Zeit müssen die erwarteten Daten empfangen sein
			//es werden nur Daten zwischen bzw. incl. STX und ETX empfangen
			//das Checksumbyte wird anschließend separat empfangen 
			fbReceiveData(pPrefix:= ADR(nPrefix),	//STX
						LenPrefix:= 1, 
						pSuffix:= ADR(nSuffix),	 //ETX
						LenSuffix:= 1, 
						pReceiveData:= ADR(aReceiveData), 
						SizeReceiveData:= SIZEOF(aReceiveData), 
						RXbuffer:= SerialPort.P_RxBuffer,
						Reset:= FALSE);
						
			IF fbReceiveData.Error > 0 THEN
				bError := TRUE;
				bBusy := FALSE;
				nErrorId := INT_TO_UINT(fbReceiveData.Error);
				nState := 99;
				RETURN;
			END_IF

			IF fbReceiveData.DataReceived THEN
				timer1(IN:= FALSE);	
				IF fbReceiveByte.Error > 0 THEN
					bError := TRUE;
					bBusy := FALSE;
					nErrorId := INT_TO_UINT(fbReceiveByte.Error);
					nState := 99;
					RETURN;
				END_IF
				nState := 5; //weiter zu ChecksumByte empfangen				
			END_IF
			
			IF timer1.Q THEN	//Timeout -> Error
				fbReceiveData(Reset:=TRUE, pReceiveData:= ADR(aReceiveData), RXbuffer:= SerialPort.P_RxBuffer);
				nErrorId := E_ErrorIdDiluter.ERRORID_ComTimeout;
				bError := TRUE;
				bBusy := FALSE;
				nState := 99;
				RETURN;
			END_IF
		
		5:	//Checksum-Byte empfangen
			fbReceiveByte(ReceivedByte=> nCheckSum, RxBuffer:= SerialPort.P_RxBuffer);
			IF fbReceiveByte.ByteReceived THEN	//Checksumbyte wurde empfangen
				SerialPort.M_ClearRxComBuffer(); //Restlichen Buffer löschen
				//#################Checksumme überprüfen###################
				nLenData := UDINT_TO_USINT(fbReceiveData.LenReceiveData);	//Länge der empfangenen Daten (zwischen bzw. incl. STX und ETX)
				
				IF NOT (F_GetCheckSumByte(aReceiveData, nLenData) = nCheckSum) THEN	//Checksumerror
					nErrorId := E_ErrorIdDiluter.ERRORID_CecksumError;
					bError := TRUE;
					bBusy := FALSE;
					nState := 99;
					RETURN;
				ELSE
					//# # # # # # # # # # # # # # # # # empfangene Daten auswerten bzw extrahieren # # # # # # # # # # # # # # # # # # # # # # # # #
					//Statusbit aus Byte2 extrahieren (Bit 5) -> Beschreibung Tecan
					bStatus := ((aReceiveData[2] AND 16#20) =  16#20);
					
					//ErrorCode aus Byte2 extrahieren (Bit 0-3) -> Beschreibung Tecan
					nErrorId := (aReceiveData[2] AND 16#0F); //Fehlercode vom Diluter
					
					//Datenblock extrahieren - stehen ab Byte 3, wenn Datenlänge größer als 4 Byte
					nLenDatablock := nLenData - 4;
					IF nLenDatablock > 0 THEN	//Daten vorhanden
						bDataIsNumeric := TRUE;
						//Beginnend mit DataByte1 (Byte3) in nData schieben
						sReceiveData := '';
						FOR i:= 3 TO (nLenDatablock + 2) BY 1 DO
							IF NOT (aReceiveData[i] >= 16#30 AND aReceiveData[i] <= 16#39) THEN	//Inhalt dieses Bytes ist nicht numerisch
								bDataIsNumeric := FALSE;	//Output zur Weiterverarbeitung, dass sReceiveData nicht numerisch 
							END_IF
							sChar := CHR(aReceiveData[i]);
							sReceiveData := CONCAT(sReceiveData,sChar);
						END_FOR
					END_IF
					bBusy := FALSE;
					nState:= 80;	//FB ready				
			
					//Diluter-Fehlercode in eigene Fehlercode umsetzen
					//an dieser Stelle kann "nErrorId" nur den Diluter-Fehlercode enthalten 
					IF nErrorId > 0 THEN
						CASE nErrorId OF
							1:	//Error beim Initialisieren
								nErrorId := E_ErrorIdDiluter.ERRORID_InitError;
							2:	//Ungültiges Kommando übergeben
								nErrorId := E_ErrorIdDiluter.ERRORID_InvalidCommand;
							3:	//Fehlerhaften Parameter übergeben
								nErrorId := E_ErrorIdDiluter.ERRORID_InvalidOperand;
							4:	//Fehlerhafte Kommandostruktur
								nErrorId := E_ErrorIdDiluter.ERRORID_InvalidCommandSeq;
							6:	//EEPROM Fehler
								nErrorId := E_ErrorIdDiluter.ERRORID_EepromFailure;
							7:	//Diluter nicht initialisiert
								nErrorId := E_ErrorIdDiluter.ERRORID_NotIniialized;
							9:	//Kolben blockiert
								nErrorId := E_ErrorIdDiluter.ERRORID_PlungerOverload;
							10:	//Ventil blockiert
								nErrorId := E_ErrorIdDiluter.ERRORID_ValveOverload;
							11:	//Kolbenbewegung nicht erlaubt
								nErrorId := E_ErrorIdDiluter.ERRORID_PlungerMoveNotAllowed;
							15:	//vorherige aktion noch nicht abgearbeitet (StatusBit noch FALSE)
								nErrorId := E_ErrorIdDiluter.ERRORID_CommandOverflow;
						END_CASE
						bError := TRUE;
						bBusy := FALSE;
						nState := 99;
					END_IF					
				END_IF
			END_IF		
	END_CASE	
ELSE
	IF SerialPort.M_IsMyTurn(THIS) THEN
		fbReceiveData(Reset:=TRUE, pReceiveData:= ADR(aReceiveData), RXbuffer:= SerialPort.P_RxBuffer);
		SerialPort.M_Release(THIS);
	END_IF
	bBusy := FALSE;
	bError := FALSE;
	nErrorId := 0;
	nState := 0;
	timer1(IN:= FALSE);
	bFlag := TRUE;
END_IF

METHOD FB_init : BOOL
VAR_INPUT
	bInitRetains : BOOL; // if TRUE, the retain variables are initialized (warm start / cold start)
	bInCopyCode : BOOL;  // if TRUE, the instance afterwards gets moved into the copy code (online change)
	SerialPort 	: REFERENCE TO FB_SerialComPort_Base;
END_VAR
THiS^.SerialPort REF= SerialPort;
END_METHOD

END_FUNCTION_BLOCK

// ---- Hardware/RS232/FB_SerialComPort_Base.TcPOU
FUNCTION_BLOCK FB_SerialComPort_Base
VAR_INPUT
END_VAR
VAR_OUTPUT
	bIsWorking 	: BOOL;
	bIsLocked	: BOOL;
END_VAR
VAR
	RxBufferSerialCom  	: Tc2_SerialCom.ComBuffer;
	TxBufferSerialCom  	: Tc2_SerialCom.ComBuffer;
	fbClearComBuffer	: Tc2_SerialCom.ClearComBuffer;
	fbFifo				: FB_SimpleFIFO_PVOID;
	bLock				: BOOL;
	rTrig				: R_TRIG;
	timerLock			: TON;
END_VAR

timerLock();
IF timerLock.Q THEN
	timerLock(IN:= FALSE);
	bIsLocked := FALSE;
END_IF

METHOD M_ClearRxComBuffer
VAR_INPUT
END_VAR
fbClearComBuffer(buffer := RxBufferSerialCom);
END_METHOD

METHOD M_ClearTxComBuffer
VAR_INPUT
END_VAR
fbClearComBuffer(buffer := TxBufferSerialCom);
END_METHOD

METHOD M_IsMyTurn : BOOL
VAR_INPUT
	pInstance : PVOID;
END_VAR
M_IsMyTurn := fbFifo.M_GetHead() = pInstance;
END_METHOD

METHOD M_LockForTime
VAR_INPUT
	tLockTime : TIME;
END_VAR
timerLock.IN := TRUE;
timerLock.PT := tLockTime;
bIsLocked := TRUE;
END_METHOD

METHOD M_Register : BOOL
VAR_INPUT
	pInstance : PVOID;
END_VAR
M_Register := fbFifo.M_Add(pInstance);
END_METHOD

METHOD M_Release : BOOL
VAR_INPUT
	pInstance : PVOID;
END_VAR
M_Release := fbFifo.M_Remove(pInstance);
END_METHOD

PROPERTY P_RxBuffer : REFERENCE TO Tc2_SerialCom.ComBuffer
GET
P_RxBuffer REF= RxBufferSerialCom;
END_GET
END_PROPERTY

PROPERTY P_TxBuffer : REFERENCE TO Tc2_SerialCom.ComBuffer
GET
P_TxBuffer REF= TxBufferSerialCom;
END_GET
END_PROPERTY

END_FUNCTION_BLOCK

// ---- Hardware/RS232/FB_SimpleFIFO_PVOID.TcPOU
FUNCTION_BLOCK FB_SimpleFIFO_PVOID
VAR_INPUT
END_VAR
VAR_OUTPUT
END_VAR
VAR
	aPool 	: ARRAY[0..15] OF PVOID;
	nList 	: ULINT; //aus diesen 64bit werden jeweils 4bit für einen Eintrag benötigt
	nCount 	: USINT;
END_VAR

//Dieser FB bietet eine schnelle und schlanke FIFO mit maximal 16 Einträgen an.

METHOD M_Add : BOOL
VAR_INPUT
	pValue : PVOID;
END_VAR

VAR
	i : USINT;
	nFreeIndex : USINT := 255;
	bAlreadyRegistered : BOOL;
END_VAR
IF pValue = 0 THEN
	RETURN;
END_IF
//Ein bereits registrierten Eintrag nicht nochmal eingetragen.
//--> Das komplette Array durchlaufen den Index merken, wo was frei ist.
FOR i := 0 TO 15 BY 1 DO
	IF aPool[i] = 0 AND nFreeIndex = 255 THEN
		nFreeIndex := i;
	ELSIF aPool[i] = pValue THEN //Eintrag bereits vorhanden -> alles abbrechen
		RETURN;
	END_IF
END_FOR

IF nFreeIndex < 255 THEN
	//Liste um ein Nibble nach links schieben
	nList := SHL(nList,4);
	nList := nList OR nFreeIndex;
	nCount := nCount + 1;
	aPool[nFreeIndex] := pValue;
	M_Add := TRUE;
END_IF
END_METHOD

METHOD M_GetHead : PVOID
VAR_INPUT
END_VAR

VAR
	nIndex : USINT;
END_VAR
IF nCount > 0 THEN
	nIndex := ULINT_TO_USINT(SHR(nList, (nCount-1)*4));
	M_GetHead := aPool[nIndex];
END_IF
END_METHOD

METHOD M_Remove : BOOL
VAR_INPUT
	pValue : PVOID;
END_VAR

VAR
	i : USINT;
	j : USINT;
	nTemp : ULINT;
	nShifts : USINT;
	nFillNibble : ULINT;
END_VAR
IF pValue = 0 THEN
	RETURN;
END_IF
FOR i := 0 TO 15 BY 1 DO
	IF aPool[i] = pValue THEN
		//nach Nibble suchen, welches den Index enthält (aber immer innerhalb der nCount-Grenzen	
		//solange nach rechts verschieben, bis LSN (lowest significat nibble) = i ist
		//danach wieder nach links verschieben, aber eins weniger
		FOR j := 0 TO nCount - 1 BY 1 DO
			nTemp := SHR(nList,((j)*4));
			IF (nTemp AND 16#F) = i THEN
				nTemp := SHR(nTemp,4);
				nTemp := SHL(nTemp,j*4);
				nShifts := (16-j)*4;
				nList := nList AND nFillNibble;
				nList := nList OR nTemp;
				aPool[i] := 0;
				nCount := nCount - 1;
				M_Remove := TRUE;
				RETURN;
			END_IF
			nFillNibble := SHL(nFillNibble,4);
			nFillNibble := nFillNibble OR 16#F;
		END_FOR
	END_IF
END_FOR
END_METHOD

END_FUNCTION_BLOCK

// ---- Hardware/Diluter/F_GetCheckSumFromString.TcPOU
FUNCTION F_GetCheckSumFromString : BYTE
VAR_INPUT
	Data	: STRING[100];	//String, aus dem die Checksumme gebildet werden soll
END_VAR
VAR
	nLenStr		:INT;		(*Länge Eingangsstring*)
	sTemp		:STRING;
	nTemp		:BYTE := 0;
	i			:INT; 	(*allg. Zählvariable*)	
END_VAR

nLenStr := LEN(Data);	//Länge des Strings

FOR i := 1 TO nLenStr BY 1 DO
	sTemp := MID(STR:= Data, LEN:= 1, POS:= i );
	nTemp := USINT_TO_BYTE(ASC(sTemp)) XOR nTemp;
END_FOR

F_GetCheckSumFromString := nTemp;

END_FUNCTION

// ---- Hardware/Diluter/F_GetCheckSumByte.TcPOU
FUNCTION F_GetCheckSumByte : BYTE
VAR_INPUT
	aData: ARRAY[0..30] OF BYTE;
	nLength: USINT;
END_VAR
VAR
	i: USINT;
	nTemp: BYTE;
END_VAR

FOR i:= 0 TO nLength-1 BY 1 DO
	nTemp := aData[i] XOR nTemp;
END_FOR

F_GetCheckSumByte := nTemp;

END_FUNCTION

// ---- Hardware/Diluter/FB_Dil_GetValveConfig.TcPOU
FUNCTION_BLOCK FB_Dil_GetValveConfig
VAR_INPUT
	bExecute	: BOOL;	
END_VAR
VAR_OUTPUT
	bBusy		: BOOL;
	bError		: BOOL;
	nErrorId	: ERRORID;
	nValue		: USINT;
END_VAR
VAR
END_VAR
VAR_IN_OUT
	DilSendCmd 	: FB_Dil_SendCmd;
	pDilRef		: POINTER TO FB_HwRefDiluter;
END_VAR

IF pDilRef = 0 THEN
	bError := TRUE;
	RETURN;	
END_IF

IF bExecute THEN
	bBusy := TRUE;

	DilSendCmd(bExecute:= TRUE, bExpectReply:= TRUE, sSendData:= CONCAT(USINT_TO_STRING(pDilRef^.nChannel),'?21'));
	
	IF NOT DilSendCmd.bBusy THEN
		IF DilSendCmd.bError THEN
			bError := TRUE;
			nErrorId := DilSendCmd.nErrorId;
		ELSE
			nValue := F_ToASC(LEFT(DilSendCmd.sReceiveData,1)) AND 16#0F;
			pDilRef^.eValveType := nValue;
		END_IF
		DilSendCmd(bExecute:= FALSE);
		bBusy := FALSE;
	END_IF
ELSE
	DilSendCmd(bExecute:= FALSE);
	bBusy := FALSE;
	bError := FALSE;
	nErrorId := 0;
	nValue := 0;
END_IF

END_FUNCTION_BLOCK

// ---- Hardware/Diluter/FB_Dil_SetValveConfig.TcPOU
FUNCTION_BLOCK FB_Dil_SetValveConfig
VAR_INPUT
	bExecute	: BOOL;
	eValveType  : E_DilValveType;
END_VAR
VAR_OUTPUT
	bBusy		: BOOL;
	bError		: BOOL;
	nErrorId	: ERRORID;
END_VAR
VAR
	nState		: USINT;
	sSendData	: STRING(100);
	timer		: TON;
END_VAR
VAR_IN_OUT
	DilSendCmd 	: FB_Dil_SendCmd;
	pDilRef		: POINTER TO FB_HwRefDiluter;
END_VAR

IF pDilRef = 0 THEN
	bError := TRUE;
	RETURN;	
END_IF

IF bExecute THEN
	CASE nState OF
		0:	//Write valve config
			bBusy := TRUE;
			sSendData := CONCAT(USINT_TO_STRING(pDilRef^.nChannel),'U');
			sSendData := CONCAT(sSendData,USINT_TO_STRING(eValveType));
			sSendData := CONCAT(sSendData,'R');
			DilSendCmd(bExecute:= TRUE, bExpectReply:= TRUE, sSendData:= sSendData);
			
			IF NOT DilSendCmd.bBusy THEN
				IF DilSendCmd.bError THEN
					bBusy := FALSE;
					bError := TRUE;
					nErrorId := DilSendCmd.nErrorId;
				ELSE
					nState := 1;
				END_IF
				DilSendCmd(bExecute:= FALSE);
			END_IF
		
		1:	//Reset
			sSendData := CONCAT(USINT_TO_STRING(pDilRef^.nChannel),'!R');
			DilSendCmd(bExecute:= TRUE, bExpectReply:= FALSE, sSendData:= sSendData);
			IF NOT DilSendCmd.bBusy THEN
				IF DilSendCmd.bError THEN
					bBusy := FALSE;
					bError := TRUE;
					nErrorId := DilSendCmd.nErrorId;
				ELSE
					nState := 2;
				END_IF
				DilSendCmd(bExecute:= FALSE);
			END_IF
		
		2:	//200ms warten, bis Diluter wieder bereit
			timer(IN:= TRUE, PT:=T#200MS);
			IF timer.Q THEN
				timer(IN:= FALSE);
				nState := 80;
				bBusy := FALSE;
			END_IF
	END_CASE
ELSE
	DilSendCmd(bExecute:= FALSE);
	bBusy := FALSE;
	bError := FALSE;
	nErrorId := 0;
	nState := 0;
END_IF

END_FUNCTION_BLOCK

// ---- Hardware/Diluter/FB_Dil_GetValvePos.TcPOU
FUNCTION_BLOCK FB_Dil_GetValvePos
VAR_INPUT
	bExecute	: BOOL;
	pDilRef		: POINTER TO FB_HwRefDiluter;
END_VAR
VAR_OUTPUT
	bBusy		: BOOL;
	bError		: BOOL;
	nErrorId	: ERRORID;
	nValue		: SINT;
	bStatus		: BOOL;
END_VAR
VAR
	sString		: STRING;
	rTrig 		: R_TRIG;
	pDilRefIntern : POINTER TO FB_HwRefDiluter;	
END_VAR
VAR_IN_OUT
	DilSendCmd 	: FB_Dil_SendCmd;
END_VAR

rTrig(CLK:= bExecute);
IF rTrig.Q THEN
	IF pDilRef = 0 THEN
		bError := TRUE;
		RETURN;	
	ELSE
		pDilRefIntern := pDilRef;
	END_IF	
END_IF

IF bExecute THEN
	bBusy := TRUE;

	DilSendCmd(bExecute:= TRUE, bExpectReply:= TRUE, sSendData:= CONCAT(USINT_TO_STRING(pDilRefIntern^.nChannel),'?6'));
	
	IF NOT DilSendCmd.bBusy THEN
		IF DilSendCmd.bError THEN
			bError := TRUE;
			nErrorId := DilSendCmd.nErrorId;
		ELSE
				nValue := 0;
			IF DilSendCmd.bDataIsNumeric THEN
				nValue := STRING_TO_SINT(DilSendCmd.sReceiveData);
			ELSE
				sString := F_ToUCase(DilSendCmd.sReceiveData);
				IF sString = 'I' THEN
					nValue := 1;
				ELSIF sString = 'O' THEN
					nValue := 2;
				ELSIF sString = 'B' THEN
					nValue := 3;
				ELSIF sString = 'E' THEN
					nValue := 4;
				END_IF
			END_IF
			pDilRefIntern^.nActValvePos := nValue;
			bStatus := DilSendCmd.bStatus;
		END_IF
		DilSendCmd(bExecute:= FALSE);
		bBusy := FALSE;
	END_IF
ELSE
	bBusy := FALSE;
	bError := FALSE;
	nErrorId := 0;
	nValue := 0;
	bStatus := FALSE;
END_IF

END_FUNCTION_BLOCK

// ---- Hardware/Diluter/FB_Dil_Init.TcPOU
FUNCTION_BLOCK FB_Dil_Init
VAR_INPUT
	bExecute	: BOOL;
END_VAR
VAR_OUTPUT
	bBusy		: BOOL;
	bError		: BOOL;
	nErrorId	: ERRORID;
END_VAR
VAR
	nState		: USINT;
	bStatus		: BOOL;
	nReadValue	: UINT;
END_VAR
VAR_IN_OUT
	DilSendCmd 	: FB_Dil_SendCmd;
	pDilRef		: POINTER TO FB_HwRefDiluter;
END_VAR

IF pDilRef = 0 THEN
	bError := TRUE;
	RETURN;	
END_IF

IF bExecute THEN
	CASE nState OF
		0:	//Status abrufen
			pDilRef^.bBusy := bBusy := TRUE;
			pDilRef^.bIsInit := FALSE;
			DilSendCmd(bExecute:= TRUE, bExpectReply:= TRUE, sSendData:= CONCAT(USINT_TO_STRING(pDilRef^.nChannel),'Q'));
			IF NOT DilSendCmd.bBusy THEN
				IF DilSendCmd.bError THEN
					bError := TRUE;
					nErrorId := DilSendCmd.nErrorId;
				ELSE
					IF DilSendCmd.bStatus THEN //ready
						nState := 2;
					ELSE //busy -> stoppen
						nState := 1;
					END_IF
				END_IF
				DilSendCmd(bExecute:= FALSE);
			END_IF

		1:	//Diluter stoppen
			DilSendCmd(bExecute:= TRUE, bExpectReply:= TRUE, sSendData:= CONCAT(USINT_TO_STRING(pDilRef^.nChannel),'T'));
			IF NOT DilSendCmd.bBusy THEN
				IF DilSendCmd.bError THEN
					bError := TRUE;
					nErrorId := DilSendCmd.nErrorId;
				ELSE
					nState := 0; //nochmal Status abrufen
				END_IF
				DilSendCmd(bExecute:= FALSE);
			END_IF
		
		2: //Init ausführen
			DilSendCmd(bExecute:= TRUE, bExpectReply:= TRUE, sSendData:= CONCAT(USINT_TO_STRING(pDilRef^.nChannel),'ZN1R'));
			IF NOT DilSendCmd.bBusy THEN
				IF DilSendCmd.bError THEN
					bError := TRUE;
					nErrorId := DilSendCmd.nErrorId;
				ELSE
					nState := 3;
				END_IF
				DilSendCmd(bExecute:= FALSE);
			END_IF
		
		3: //Status abrufen
			DilSendCmd(bExecute:= TRUE, bExpectReply:= TRUE, sSendData:= CONCAT(USINT_TO_STRING(pDilRef^.nChannel),'Q'));
			IF NOT DilSendCmd.bBusy THEN
				IF DilSendCmd.bError THEN
					bError := TRUE;
					nErrorId := DilSendCmd.nErrorId;
				ELSE
					IF DilSendCmd.bStatus THEN
						pDilRef^.bBusy := bBusy := FALSE;
						pDilRef^.bIsInit := TRUE;
						nState := 80;
					END_IF
				END_IF
				DilSendCmd(bExecute:= FALSE);
				
			END_IF
	END_CASE
	
	IF bError THEN
		pDilRef^.bBusy := bBusy := FALSE;
		nState := 99;
	END_IF
ELSE
	DilSendCmd(bExecute:= FALSE);
	nState := 0;
	pDilRef^.bBusy := bBusy := FALSE;
	bError := FALSE;
	nErrorId := 0;
END_IF

END_FUNCTION_BLOCK

// ---- Hardware/Diluter/FB_Dil_Transfer.TcPOU
FUNCTION_BLOCK FB_Dil_Transfer
VAR_INPUT
	pDilRef1		: POINTER TO FB_HwRefDiluter;
	pDilRef2		: POINTER TO FB_HwRefDiluter;
	nTransferSteps	: UDINT;	//TransferMenge in Microsteps
	nPreSteps		: INT;
	nPostSteps		: INT;
	nValveInput1	: SINT;		//Ventilstellung Input(SystemLiquid) Source (Press-Diluter)
	nValveOutput1	: SINT;		//Ventilstellung Output(Luer) Source (Press-Diluter)
	nValveWaste1	: SINT;		//Ventilstellung Waste Source (Press-Diluter)
	nValveInput2	: SINT;		//Ventilstellung Input(SystemLiquid) Source (Suck-Diluter)
	nValveOutput2	: SINT;		//Ventilstellung Output(Luer) Source (Suck-Diluter)
	nValveWaste2	: SINT;		//Ventilstellung Waste Source (Press-Diluter))*)
	nSpeedPump		: DINT;		//Gechwindigkeit Pumpen in Halbsteps/s
	nSpeedReload	: DINT;		//Gechwindigkeit Nachladen in Halbsteps/s
	bExecute		: BOOL;
END_VAR
VAR_OUTPUT
	bBusy		: BOOL;
	bError		: BOOL;
	nErrorId	: ERRORID;
END_VAR
VAR
	rTrig 				: R_TRIG;
	nState				: USINT;
	sString				: STRING[100];	//Sendestring
	sValvePos			: STRING[2];
	sValvePos2			: STRING[2];
	nStartPosSrc		: UINT;
	nStartPosDest		: UINT;
	nCurPlungerPosSrc	: UINT;
	nCurPlungerPosDest	: UINT;
	nTotalSteps			: UDINT;
	
	pDilRefSrc			: POINTER TO FB_HwRefDiluter;
	pDilRefDest			: POINTER TO FB_HwRefDiluter;
	nValveInputSrc		: SINT;		//Ventilstellung Input(SystemLiquid) Source (Press-Diluter)
	nValveOutputSrc		: SINT;		//Ventilstellung Output(Luer) Source (Press-Diluter)
	nValveWasteSrc		: SINT;		//Ventilstellung Waste Source (Press-Diluter)
	nValveInputDest		: SINT;		//Ventilstellung Input(SystemLiquid) Source (Suck-Diluter)
	nValveOutputDest	: SINT;		//Ventilstellung Output(Luer) Source (Suck-Diluter)
	nValveWasteDest		: SINT;		//Ventilstellung Waste Source (Press-Diluter))*)
	
	fbGetPlungerPos		: FB_Dil_GetPlungerPos;
	fbGetValvePos		: FB_Dil_GetValvePos;
	fbMoveToPos			: FB_Dil_MoveToPos;
END_VAR
VAR_IN_OUT
	DilSendCmd 	: FB_Dil_SendCmd;
END_VAR

rTrig(CLK:= bExecute);
IF rTrig.Q THEN
	IF pDilRef1 = 0 OR pDilRef2 = 0 THEN
		bError := TRUE;
		RETURN;	
	ELSE
		pDilRefSrc := pDilRef1;
		nValveInputSrc := nValveInput1;
		nValveOutputSrc := nValveOutput1;
		nValveWasteSrc := nValveWaste1;
		pDilRefDest := pDilRef2;
		nValveInputDest := nValveInput2;
		nValveOutputDest := nValveOutput2;
		nValveWasteDest := nValveWaste2;
	END_IF	
END_IF

(*Diluter in jeweilige Ausgangsstellung fahren:
Es gibt 3 verschiedene Möglichkeiten
1. 	PreSteps > 0: 
   	DilPress beginnt früher -> DilPress: Bottom, DilSuck: Top - PreSteps
	DilSuck startet mit Delay
2. 	PreSteps = 0:
	Beide starten zugeleich -> DilPress: Bottom, DilSuck: Top
3.	PreSteps < 0:
	DilSuck beginnt früher -> DilPress: Bottom + PreSteps, DilSuck: Top
	DilPress startet mit Delay
*)

IF bExecute THEN
	IF nState = 0 THEN	//Aktuelle Kolbenposition DilSrc abrufen
		bBusy := TRUE;
		fbGetPlungerPos(DilSendCmd:= DilSendCmd, pDilRef:= pDilRefSrc, bExecute:= TRUE);
		IF NOT fbGetPlungerPos.bBusy THEN
			IF fbGetPlungerPos.bError THEN
				bError := TRUE;
				nErrorId := fbGetPlungerPos.nErrorId;
				bBusy := FALSE;
			ELSE
				nCurPlungerPosSrc := fbGetPlungerPos.nValue;
				nState := 1;
			END_IF
			fbGetPlungerPos(DilSendCmd:= DilSendCmd, bExecute:= FALSE);
		ELSE
			RETURN;
		END_IF
	END_IF
	
	IF nState = 1 THEN	//Aktuelle Kolbenposition DilDest abrufen
		fbGetPlungerPos(DilSendCmd:= DilSendCmd, pDilRef:= pDilRefDest, bExecute:= TRUE);
		IF NOT fbGetPlungerPos.bBusy THEN
			IF fbGetPlungerPos.bError THEN
				bError := TRUE;
				nErrorId := fbGetPlungerPos.nErrorId;
				bBusy := FALSE;
			ELSE
				nCurPlungerPosDest := fbGetPlungerPos.nValue;
				//Startpositionen berechenen
				IF nPreSteps > 0 THEN
					nStartPosSrc := 24000;
					nStartPosDest := INT_TO_UINT(nPreSteps);
				ELSIF nPreSteps = 0 THEN
					nStartPosSrc := 24000;
					nStartPosDest := 0;
				ELSE // < 0
					nStartPosSrc := INT_TO_UINT(24000 + nPreSteps);
					nStartPosDest := 0;
				END_IF
				nState := 2;
			END_IF
			fbGetPlungerPos(bExecute:= FALSE, DilSendCmd:= DilSendCmd);
		ELSE
			RETURN;
		END_IF
	END_IF
	
	IF nState = 2 THEN	//Startposition DilSrc anfahren
		sString := CONCAT(USINT_TO_STRING(pDilRefSrc^.nChannel),'v100c100V');	//Startspeed,CutOffSpeed + Kennung für Topspeed
		sString := CONCAT(sString,DINT_TO_STRING(nSpeedReload));		//Topspeed
		//Ventilstellung ist abhängig von aktueller Kolbenposition
		IF nStartPosSrc < nCurPlungerPosSrc THEN //Drücken in Waste
			sValvePos := F_GetValveCode(nValveWasteSrc,pDilRefSrc^.nActValvePos,pDilRefSrc^.eValveType);
			sString := CONCAT(sString,sValvePos);					//Ventilstellung in Richtung Waste	
		ELSE //Saugen aus Input
			sValvePos := F_GetValveCode(nValveInputSrc,pDilRefSrc^.nActValvePos,pDilRefSrc^.eValveType);
			sString := CONCAT(sString,sValvePos);					//Ventilstellung in Richtung Input(SystemLiquid)
		END_IF
		IF sValvePos = '' THEN
			bError := TRUE;
			nErrorId := E_ErrorIdDiluter.ERRORID_InvalidValveParam;
			RETURN;
		END_IF
		sString := CONCAT(sString,'A');									//Kennung für Move
		sString := CONCAT(sString, UINT_TO_STRING(nStartPosSrc));		//Position
		sValvePos := F_GetValveCode(nValveOutputSrc,pDilRefSrc^.nActValvePos, pDilRefSrc^.eValveType);
		IF sValvePos = '' THEN
			bError := TRUE;
			nErrorId := E_ErrorIdDiluter.ERRORID_InvalidValveParam;
			RETURN;			
		END_IF
		sString := CONCAT(sString,sValvePos);						//Ventilstellung in Richtung Luer nach Erreichen Startposition
		sString := CONCAT(sString,'R');									//Execute-Zeichen
		
		DilSendCmd(bExecute:= TRUE, bExpectReply:= TRUE, sSendData:= sString);
		
		IF NOT DilSendCmd.bBusy THEN
			IF DilSendCmd.bError THEN
				bError := TRUE;
				nErrorId := DilSendCmd.nErrorId;
				bBusy:= FALSE;
			ELSE
				nState := 3;
			END_IF
			DilSendCmd(bExecute:= FALSE);
		ELSE
			RETURN;
		END_IF
	ELSIF nState = 3 THEN	//Startposition DilDest anfahren
		sString := CONCAT(USINT_TO_STRING(pDilRefDest^.nChannel),'v100c100V');	//Startspeed,CutOffSpeed + Kennung für Topspeed
		sString := CONCAT(sString,DINT_TO_STRING(nSpeedReload));		//Topspeed
		//Ventilstellung ist abhängig von aktueller Kolbenposition
		IF nStartPosDest < nCurPlungerPosDest THEN //Drücken in Waste
			sValvePos := F_GetValveCode(nValveWasteDest,pDilRefDest^.nActValvePos,pDilRefDest^.eValveType);
			sString := CONCAT(sString,sValvePos);					//Ventilstellung in Richtung Waste	
		ELSE //Saugen aus Input
			sValvePos := F_GetValveCode(nValveInputDest,pDilRefDest^.nActValvePos,pDilRefDest^.eValveType);
			sString := CONCAT(sString,sValvePos);					//Ventilstellung in Richtung Input(SystemLiquid)	
		END_IF
		
		IF sValvePos = '' THEN
			bError := TRUE;
			nErrorId := E_ErrorIdDiluter.ERRORID_InvalidValveParam;
			RETURN;
		END_IF		
		sString := CONCAT(sString,'A');									//Kennung für Move
		sString := CONCAT(sString, UINT_TO_STRING(nStartPosDest));		//Position
		sValvePos := F_GetValveCode(nValveOutputDest,pDilRefDest^.nActValvePos, pDilRefDest^.eValveType);
		IF sValvePos = '' THEN
			bError := TRUE;
			nErrorId := E_ErrorIdDiluter.ERRORID_InvalidValveParam;
			RETURN;			
		END_IF		
		sString := CONCAT(sString,sValvePos);						//Ventilstellung in Richtung Luer nach Erreichen Startposition
		sString := CONCAT(sString,'R');							//Execute-Zeichen
		
		DilSendCmd(bExecute:= TRUE, bExpectReply:= TRUE, sSendData:= sString);
		
